	arRauschen: ARRAY [0..9999] OF REAL := [0.246739256236, -0.529170105611, 0.414309825378, -0.544103926825, 0.009949783811, -0.029587575492, -0.961653654724, -0.382605463343, 0.222026883158, 0.389023823093, 0.621050671571, -0.646958412688, 0.638418207627, 0.534061065662, -0.110754415353, 0.629669607832, -0.372363722573, -0.871060345803, 0.681706748020, 0.205129983440, 0.858041542734, -0.075593969433, -0.319802679147, 0.977319730903, -0.463662632934, 0.393306864076, -0.217856355895, -0.964407875275, 0.809210531413, 0.985531542521, -0.674619330252, 0.436784775739, -0.160868201578, 0.341967854837, -0.399787326721, 0.290907556563, 0.539355132357, -0.823844250498, -0.040486992077, 0.198136927055, -0.108719761440, -0.795757664573, -0.924329592637, 0.258815633556, -0.272619658361, 0.669346919862, 0.120580060721, -0.412226444472, -0.863110760094, 0.848406544850, -0.407508257473, -0.683558789495, -0.591427504389, 0.316833250828, -0.966288801701, -0.227470576788, 0.579664019389, -0.594067152985, -0.737773981554, 0.224918962597, -0.702529720677, 0.652896341734, -0.876627290498, 0.775098206896, -0.335284108258, 0.727377951755, -0.229819698701, 0.541187889029, -0.041203903558, -0.635223979412, -0.016835900977, -0.081127400735, 0.473800100213, 0.370010232427, -0.781292715531, 0.151475020756, -0.928262298559, 0.719073235463, 0.944742409840, 0.859713266715, -0.234696976409, 0.466709694464, 0.972663248100, -0.093433859902, -0.240648257108, 0.600574830997, -0.676848255859, -0.664059236041, -0.772492529238, -0.525769140900, -0.445967976269, -0.422592640425, -0.817647930030, 0.622493353226, 0.969345965405, 0.749765014787, -0.941528041560, 0.567473529861, 0.330423592919, 0.628163921603, 0.865778023332, -0.925525550689, 0.250234639214, 0.178032614233, 0.845317953168, -0.724431653562, 0.326294937160, -0.998925438332, -0.144238934713, 0.936006148019, 0.028752943103, -0.007566843574, -0.657885652494, -0.544697262441, 0.431807667642, -0.115466610367, 0.644197371225, -0.473158752747, -0.104897086620, -0.557304583420, -0.693084284084, -0.266431314125, -0.657718817527, 0.012733837449, -0.356939242672, -0.582847192411, -0.321250664899, -0.000437913139, -0.801730193481, -0.395392715595, 0.753309159993, -0.839167873710, -0.497709637142, 0.376142374662, -0.891710910001, -0.931460999004, -0.765244974856, -0.430077335395, -0.165793475662, -0.067370896287, 0.716185225145, 0.093961060499, -0.600848329188, 0.673058447165, 0.674704320685, -0.027227232800, 0.171745340627, -0.918910173725, 0.209163411102, 0.680797609799, 0.067226768430, -0.999009889300, -0.780625702217, 0.367241297318, 0.402204046803, 0.285102145157, 0.183271048762, 0.995194348284, -0.806487621398, 0.112997935460, -0.561176200081, 0.453177893515, -0.405486497721, -0.698964164112, -0.893396062005, 0.294927669631, -0.287540801977, -0.398405888092, 0.401119508788, -0.505326064545, -0.225827285260, -0.294225352090, 0.144798347025, -0.430384210188, 0.666149813029, 0.883918289765, 0.949635828195, 0.724396900619, 0.156010733086, 0.447585744588, 0.443566930836, 0.105623713564, 0.480873497360, 0.478874307928, -0.363553379976, -0.292587342811, 0.391116870080, 0.509282603531, 0.026478500049, 0.278623039847, 0.213444321271, -0.651644355304, -0.081057820072, -0.006698364322, 0.842760715437, 0.416093279887, -0.696197758558, -0.713828347366, -0.065887452693, 0.297891975424, 0.475395401787, -0.835706801589, -0.234477046070, -0.728620258748, 0.142537813675, -0.496592649012, 0.427164188114, -0.872643068742, 0.392931044892, -0.391015917539, -0.908629066401, -0.373314983099, -0.518141560956, -0.274306877176, 0.477171922966, -0.418180886710, -0.466110720658, 0.577632902938, 0.334027359560, -0.761070711022, -0.958568115698, 0.668176974590, 0.000497204020, 0.525722665811, -0.767668130265, -0.244392457220, 0.462184067229, -0.047276594620, 0.084864277025, -0.115062364457, -0.715907950963, 0.158290277543, 0.430925333764, -0.237143624360, -0.921853342785, -0.180352070779, 0.872419264731, -0.298218856373, 0.012398576959, -0.102073877969, -0.016164126855, 0.344215775954, 0.062456227753, -0.045480709999, -0.612235813695, 0.927440580288, 0.128274592282, 0.367175640002, 0.522036080855, -0.514356302852, 0.032995121162, 0.024509715061, 0.845448084989, 0.447884205959, 0.847428365298, -0.208174858415, -0.544927435342, -0.404805621403, -0.613620769868, -0.706941066657, 0.332305269893, -0.072931291890, -0.249740966904, -0.759240606791, -0.865256880141, 0.630348896703, -0.746062522885, -0.358926494928, 0.129871216481, 0.524777575363, 0.554834351075, 0.291634864464, 0.862406170075, -0.439019664257, -0.167620988081, 0.474524278117, -0.253399651970, -0.447962964225, 0.184329851673, 0.448599046466, -0.979074329430, 0.347509289836, 0.440450729671, -0.181101795764, 0.051759350663, -0.386345551805, 0.844407334874, -0.617550553980, 0.818452991754, 0.605805879582, -0.644762312935, -0.607126658097, -0.697909226410, -0.867331983037, -0.538829948377, 0.920977238585, 0.907194206181, 0.637867983590, 0.729978494237, 0.326346021492, -0.993639828643, -0.047669394639, -0.978448647461, -0.187853782006, -0.344460373153, -0.693377000027, 0.751878997091, 0.811489751365, 0.323523735780, 0.022615842344, -0.151697873914, 0.316030939885, -0.210096145889, -0.948333340436, -0.911576847596, 0.826438670365, -0.744203261189, 0.772633117720, 0.181996339876, 0.935860210219, -0.099340173278, -0.800545523085, 0.756346944715, 0.319694561318, 0.972386432025, 0.204278217384, 0.913860972173, 0.937730762197, 0.312294177414, -0.261802998374, -0.635043991959, -0.235704358395, 0.466866088657, 0.351908922889, 0.591241011493, 0.727184996899, -0.564588415423, 0.667864381168, 0.300950655987, -0.155187192446, -0.397009717286, -0.525668199483, -0.456722345352, -0.823156392312, 0.788091934648, -0.753677385492, 0.682613050591, 0.804545831956, -0.334143783172, 0.111262921985, -0.852217512624, -0.041248860227, 0.778424005231, 0.044092776273, -0.065148797437, -0.757446664925, 0.155584195178, -0.820895820909, 0.011012148577, 0.374346119688, -0.579777277082, 0.385402006686, -0.988425659978, 0.239650409460, 0.907806660527, 0.751302397733, -0.068518188527, 0.480588932436, -0.569440051514, 0.619651395135, 0.024224185726, -0.785251187626, -0.983163309183, -0.415107378772, 0.613246911220, -0.250774675569, 0.371154100200, -0.219976331516, -0.220820891629, 0.127276136859, 0.824871934223, -0.534679223208, -0.938731233427, 0.752572249594, -0.847763317363, -0.728473978394, -0.646685665337, -0.998230717786, -0.860355633059, 0.198309069301, 0.332641337457, -0.788086027259, 0.696356744821, -0.804116334097, -0.799940505629, 0.547771798051, -0.852007662520, 0.337985525103, -0.733625872664, 0.660112536732, -0.321721536287, 0.003955703369, 0.351169972261, -0.311372520781, 0.313518004463, -0.891545308924, 0.496612274384, -0.176333071866, 0.537443706881, -0.488325145144, 0.538839566528, 0.539455258831, 0.735078466938, -0.688582146983, 0.949128810865, 0.963534159979, -0.259586191929, -0.129749758499, 0.493600721045, -0.859039053261, 0.525898193207, -0.384840282320, 0.742109951586, 0.302311170266, -0.808430002728, 0.420777325583, 0.959985318514, -0.505694203965, 0.031473307543, -0.167052683511, 0.500995058621, -0.156240823058, -0.744660490876, -0.854345614702, 0.189686977569, 0.821968916196, 0.811848983783, -0.342248024788, 0.023386872211, -0.660481237660, -0.460544835850, 0.556515458246, -0.557324905873, -0.593178975950, -0.736410294210, 0.416696052525, -0.481910925306, -0.156710336625, -0.663890549795, 0.911054419764, -0.980908485241, -0.071421964265, 0.721864961899, 0.006623412636, 0.188458995265, 0.843334923818, -0.774386976596, -0.807321577917, 0.815744326141, -0.951120224240, -0.144390611699, -0.026540746706, -0.874864609556, 0.014619343280, -0.208958616452, 0.758626928611, -0.438345080326, 0.501296544538, -0.183694685477, 0.391828497818, -0.407011942600, -0.977859890170, -0.762130246845, -0.297107556927, -0.122704330333, -0.082888661982, -0.523983815486, -0.168575036587, -0.676178838144, 0.244686771623, -0.525082355123, -0.118407067617, 0.856705759830, 0.899986679545, 0.232731619176, -0.373659041440, -0.758853640143, -0.946684132010, 0.042597300244, -0.633489527377, 0.397335233294, 0.860053377735, -0.969386507574, -0.608982349462, 0.919627898896, 0.104498194003, -0.231531036526, 0.461295456936, -0.697220054250, 0.523414803843, -0.978859356941, -0.311641882775, -0.515670048627, 0.674862728618, -0.115816520827, 0.876629539024, -0.371659034411, 0.693339507317, 0.271248632601, 0.697480469246, 0.905967150449, 0.979868201460, 0.253258815661, -0.523955707108, 0.234763559449, -0.093833082248, -0.305544070723, -0.478107158023, -0.697737228676, 0.160904001479, -0.699222850226, -0.350695766840, -0.093324239932, 0.590288847606, -0.472075268771, -0.997304662950, -0.413944129832, 0.963282831881, -0.538669864124, -0.561804500270, 0.093857934354, -0.896970395490, 0.858943676421, 0.433641515365, -0.839191009984, 0.110506309259, -0.913682948113, -0.461490457417, 0.050243383716, -0.988280605990, 0.389764037791, 0.363904430651, 0.214157788563, 0.467709226526, 0.519997364236, 0.135818530443, 0.684759164261, -0.603702119034, -0.268419316193, 0.877117109797, 0.931384739652, -0.140717573327, 0.981671923886, -0.135246954639, -0.232401387562, 0.785244099903, -0.512140135299, 0.915155265966, 0.478784070983, -0.275938774048, -0.404748087264, 0.454006166650, 0.770802615119, 0.321755074255, -0.044838103921, -0.044766397818, 0.298751702852, -0.179385623660, 0.809437923947, -0.833841848312, 0.753779650674, -0.913838518064, -0.376044191736, -0.068730117317, -0.542593871867, -0.389049565052, -0.309568273925, 0.817561615928, -0.228143443931, 0.642328905857, -0.733360603876, 0.275236333669, 0.702112237526, 0.624421394323, 0.481857177133, 0.583799350677, -0.065337413748, 0.931548235238, -0.625969083958, -0.834512522213, -0.005650015820, -0.246010382853, 0.081298781207, 0.376488263004, 0.958702174688, -0.945974458932, -0.915934484488, -0.874287612394, 0.916799883156, -0.469450442152, 0.440713677224, 0.195323675413, 0.617040350545, -0.837318734479, 0.169952319734, 0.153771659724, 0.486478528275, -0.638819160697, 0.645997593065, -0.915354925421, -0.152165518207, 0.060295551424, 0.179416883964, -0.772015302469, 0.086118181691, -0.562826107422, -0.275447780295, 0.063906505211, -0.633526394653, -0.455850104037, -0.120851955932, 0.421106032794, 0.499620343209, -0.598850065060, -0.646616427358, 0.357237736603, -0.193854809814, 0.567724730445, 0.195663475127, -0.372821260522, -0.158056750685, -0.855837956202, 0.423096592926, 0.047027995341, -0.758922025278, 0.356971778983, 0.443647347943, -0.042147361226, 0.215564251448, 0.068340041183, 0.177291269390, -0.870104557139, 0.939236777196, 0.365008785213, 0.604158730590, -0.929579718916, -0.163665978021, -0.511346949857, 0.242462760136, -0.362591367359, 0.557188420226, -0.606221422767, 0.741195281289, 0.077036426793, 0.048193010512, 0.314666123135, -0.984858428444, 0.460746639204, 0.946057661354, -0.946166863918, 0.272900975827, -0.616788394308, 0.251179257590, 0.202353079566, -0.061445284179, -0.385572779586, -0.295799961294, -0.938227060849, -0.508337996617, 0.799743401620, -0.410014090727, 0.237535782472, 0.751036304509, -0.706447842465, -0.263237507081, -0.394747690100, -0.688150714247, -0.172462825669, -0.218692099507, -0.037766029401, -0.178199659551, -0.470927558837, 0.883228663781, 0.049918702856, 0.444438157474, 0.159857443072, 0.282221533557, 0.715223629573, 0.532428592597, -0.986489840111, -0.650364361217, 0.058543996800, -0.501009480370, -0.400235784214, -0.589280300995, 0.566421866038, 0.443685317696, -0.674411494955, 0.038062417014, 0.944215890637, 0.718572105839, -0.873071804215, -0.836357861660, 0.861249876716, 0.852403633336, 0.009361961914, 0.335102239078, 0.690320925472, -0.342135457788, 0.726486980000, -0.217484450717, -0.126917711359, -0.242431173859, 0.167341452212, 0.340963770653, -0.570551213657, -0.393229093423, -0.747032607878, -0.849476553392, 0.867814185849, 0.394966585026, -0.476517758907, 0.824517768713, -0.123745685474, -0.763511110781, 0.511435368053, -0.671460109581, -0.060036379791, -0.102884307714, 0.656986657907, -0.653404039677, 0.042770136203, 0.491850594452, 0.228272575543, 0.562898627376, 0.819041191154, 0.353312344924, 0.458881968727, -0.485155298790, 0.055094383845, -0.918719910364, -0.772592375745, 0.153732123944, -0.555993184464, 0.433087663116, 0.963410159996, 0.161010932370, -0.877731667709, 0.072961348815, 0.957803045363, -0.169325549683, -0.210430078261, 0.270182370919, 0.364976811671, 0.000887526570, 0.658057122004, 0.194342134023, 0.608790824187, -0.591578116787, -0.584628982855, -0.048320241703, 0.689196065412, -0.501091940331, -0.509502674411, 0.828689067846, -0.186360125620, 0.358118283074, -0.777402918788, -0.909671164058, 0.543782291077, 0.417043659840, -0.225356227100, -0.805139717432, 0.303729795010, 0.407044796304, -0.039811239061, 0.446407632663, 0.775584820949, -0.004740014571, 0.951315069235, 0.504543903117, -0.071948646061, -0.625458297470, -0.729660874600, 0.293493538124, 0.665903079080, -0.991178420286, 0.941126844696, -0.108546075344, 0.301003734455, -0.515422065553, -0.796223436435, 0.708593336614, -0.044071273723, -0.238737149707, -0.277276977417, -0.299167199866, -0.611572820793, 0.643683836363, -0.311036762095, 0.034698347125, -0.736555289597, -0.059452166273, -0.841744489550, -0.399957487547, 0.048641034050, 0.691121843116, -0.426142937448, 0.802617662814, -0.741494329790, -0.477954661499, 0.328158133299, -0.512215165726, -0.541295174311, -0.230194439432, -0.547034374221, -0.062024009281, 0.349314375953, -0.916724218411, -0.092744380301, -0.242786357167, -0.286735046168, -0.559148602503, 0.449041763777, -0.745158707512, -0.513680934139, 0.786026025783, -0.504750350939, 0.055350545515, 0.799483633198, 0.934405810138, 0.033922169696, 0.720637994545, 0.418491709645, 0.880158844967, -0.163137441728, 0.867818746018, -0.035334145941, -0.316515700042, -0.789617761172, -0.536104042001, -0.055134269823, -0.995597114343, -0.177001442665, 0.040769114729, 0.281875099989, 0.335676794887, -0.808991487370, -0.203335136870, 0.264173263606, 0.677808014455, -0.778769587235, -0.243410881675, -0.221057920766, -0.373071848858, -0.964506167651, 0.925577006119, -0.145365769285, -0.745957096826, -0.837329737556, -0.649573720357, -0.243767331016, -0.717820957602, -0.488103996047, 0.589287912555, -0.035391824711, 0.332107535576, 0.073973801950, 0.655044637327, -0.709540589187, -0.716071780494, -0.837772118059, -0.027656728571, -0.844827968721, -0.151940535527, -0.413167239818, 0.005011514053, -0.099245898407, 0.075226772186, 0.288592494403, -0.408640040908, 0.817498184105, -0.027674266586, -0.864782709192, 0.895092419611, 0.142483538548, 0.530743178155, -0.877081916830, 0.153623861285, 0.963376011897, -0.376765708130, 0.343760697511, -0.656038487855, 0.961393976984, 0.969850800604, 0.704099978064, -0.321644469795, -0.194963241375, -0.845246484367, 0.883097150948, 0.523139557285, -0.025904872022, -0.474928370917, 0.464591963031, -0.608894540802, 0.703450877615, -0.840748471231, 0.074940737279, -0.912829004070, 0.316523577937, 0.667685368412, -0.157405198168, 0.777038399599, 0.426964555419, 0.305664733153, -0.783179585430, -0.773095971142, -0.349441959185, 0.649764345670, -0.819401256290, 0.550662506970, 0.958334092391, -0.807662340887, 0.340864538215, 0.795147589984, -0.432285658620, -0.938935951697, 0.692164323306, -0.449196593529, -0.287304596732, 0.418878370143, 0.152337702287, -0.207140809159, 0.394871842309, 0.830431123909, 0.818073779406, -0.978273905752, -0.862804063048, -0.730298413145, 0.440110200389, -0.393436326766, -0.652877842189, 0.909220362579, 0.739095986019, -0.825817330538, -0.798492736161, 0.562865296033, 0.243296330804, -0.486844317404, -0.331653232697, -0.522004993936, -0.206970157282, -0.088377834029, 0.421952097925, -0.600802259125, 0.213859636921, 0.835919698579, 0.273560326920, -0.688558654402, 0.275055148223, 0.439068501528, 0.595496790447, 0.191442384332, -0.586591331319, 0.461177787306, 0.035502975523, -0.979483729818, 0.754914986795, 0.383257281124, -0.584778905712, 0.460985106816, -0.397540695073, -0.731321472446, 0.714271395786, 0.462776349401, 0.841844366225, -0.989997240947, -0.794638764199, -0.449690047504, -0.485538344668, -0.569066888656, -0.829496691942, -0.942956277379, 0.127429811264, 0.514096335955, -0.814996499054, -0.255271011683, 0.153170001235, 0.040702163574, -0.109755873757, 0.461556415658, -0.285080354765, -0.359789189277, 0.797148795582, 0.876352921004, 0.152166138928, -0.982440683952, 0.726129376904, -0.278422033739, 0.119560149915, 0.135627033629, -0.933593953702, 0.033842275089, -0.287177944145, 0.056212740374, 0.110418004794, 0.434676986715, 0.458408936391, 0.265619871609, 0.061257444881, -0.564588981038, 0.567841708280, -0.084344918771, -0.721688038706, 0.920242181131, 0.059390323772, -0.971319512657, -0.399220847061, -0.309027772333, -0.665363591489, -0.912709004152, -0.073862012407, 0.067684596554, -0.703681672957, -0.547543658975, -0.942830327682, 0.480511364294, 0.172985804095, 0.476793641540, 0.617990852035, -0.796430457935, 0.857861552747, 0.413594858525, 0.635925504248, -0.866751432050, -0.796863625788, -0.495670984759, -0.374977509357, 0.323023038392, -0.356534495453, -0.839284955030, 0.980838093521, -0.342406482293, -0.280793061649, 0.198936404862, 0.659048010334, 0.137553776046, 0.874818625813, -0.020766385024, 0.378235309364, 0.968067350445, 0.986534895183, -0.321368024193, -0.328216010417, 0.798171189457, 0.251190618051, -0.326446960048, 0.630696989342, 0.182914999951, -0.025160469998, 0.272208029527, 0.565919402934, 0.487738200483, -0.548172166662, -0.507209552389, -0.509070930640, -0.167269403356, -0.644923529584, 0.924804317692, -0.478564518226, -0.921762677181, -0.646762762636, -0.533560573390, -0.347591373899, 0.699635085442, -0.614636631781, 0.859517880907, -0.955001789556, 0.339146930192, 0.365286937025, 0.524010757265, -0.675270692697, 0.614162430227, 0.457875594387, -0.863092236849, -0.198092769343, -0.813516517860, 0.223903042725, -0.436347746362, 0.780841218584, 0.909398367207, -0.495892735780, 0.477911444061, -0.569395987579, -0.146650972714, -0.606544270858, 0.277434218151, -0.754911017839, 0.305274603827, 0.622224695243, -0.393998401653, -0.140010936742, -0.203988000067, -0.511531881327, -0.680583914457, 0.388166832955, 0.344343280756, -0.240779016581, 0.509725385335, -0.844520036211, -0.117103505839, 0.725892821341, 0.291263168269, 0.586311497539, -0.776273780858, 0.906667352621, 0.846415599943, 0.097490046589, 0.684382903922, -0.545299430629, 0.256859392073, -0.589408888082, -0.749586991425, -0.164804485149, -0.930954064471, -0.299620409894, 0.064335067790, -0.266619576663, 0.542000945586, -0.785794228124, 0.138801075284, 0.294517784166, 0.710127814010, 0.511363187864, -0.388462772725, 0.928953060587, -0.266970366432, 0.361628526609, -0.412034265924, -0.666934288741, 0.569230303885, 0.152134734222, 0.489457237793, 0.876157261275, 0.501140460733, 0.427246142821, 0.917589853444, 0.413867107697, -0.580480047566, 0.287150649219, 0.745621043427, 0.136538598132, 0.613800058631, -0.581144366207, -0.281306268550, 0.992292298765, -0.696688373285, 0.917588394205, -0.820359686104, -0.676661003820, -0.842408881117, -0.994234365810, -0.319103516201, -0.736723382956, -0.604760329980, 0.818239969710, 0.783820507001, 0.246185944115, -0.657196016149, -0.403697888127, -0.995150780822, 0.692288572933, 0.168061088419, 0.119921846627, 0.364989540303, -0.855680798907, -0.263656867290, -0.894865928753, 0.510699768994, 0.189185897617, -0.447285115440, -0.672978657070, 0.834544176670, 0.560712991509, -0.157172179788, 0.241893748675, -0.059960462351, 0.984749426453, 0.574429944373, -0.984005166876, -0.242616120460, -0.672194868062, -0.343482956009, 0.754578450154, -0.733255200807, -0.234196001373, 0.745137179546, 0.754168024554, 0.064314078103, -0.077932538635, -0.529696834070, 0.143181168371, 0.838996365305, -0.912757111243, 0.614893187871, -0.751880319198, 0.565478478436, -0.834012040735, 0.834466377047, 0.605493386525, 0.840176685857, 0.698476369341, -0.633077310679, 0.210397998923, -0.759788118676, 0.140552079897, 0.631965731021, -0.528836352059, -0.158802010956, 0.990369770890, -0.019803869168, -0.134520091606, 0.565686289784, -0.455613945489, 0.801903618746, -0.158640228982, 0.717202496622, -0.547831813729, 0.244780469968, -0.424876448018, 0.170836119607, 0.007398442955, 0.911729640675, 0.352723162010, -0.688599645402, -0.987557967310, 0.004866581123, 0.414027928388, -0.060997306452, 0.902315804242, 0.184449868194, -0.457073124164, -0.482700961612, 0.989282136499, 0.355302371863, 0.121561929992, 0.149376757201, 0.270869652267, -0.283803320000, 0.512882192147, -0.553083224721, -0.156770437985, -0.895244716044, -0.213404435345, 0.404663270200, -0.517802746353, -0.299143736385, 0.947496135212, 0.044415796670, 0.243940042318, -0.541746896363, 0.203075323992, -0.647373783849, 0.475455763212, 0.950029222674, -0.411124154545, 0.206910963904, -0.376899069888, -0.134490023804, -0.102678379475, -0.652690435762, -0.644841599001, 0.686166702982, 0.571332510414, -0.721995108026, -0.043151777450, -0.402344607467, 0.723838002602, -0.509802094526, 0.242244647607, 0.124710494179, -0.323613063161, -0.619797177647, 0.794161575859, 0.005887026618, 0.124043250601, 0.289828170929, 0.838632442156, 0.848401675807, 0.988685107482, 0.662462185339, 0.555603436176, 0.482507072074, -0.728481929026, 0.771618140088, 0.616755659382, 0.126330312130, -0.165651875853, 0.613194851370, 0.598795166672, 0.323378347178, 0.691073675685, 0.241795368319, 0.836520608106, 0.634843396184, -0.152796408955, 0.882721742951, -0.249667384979, 0.448022550928, -0.973888495732, -0.048223282158, -0.672215653461, -0.117773503850, -0.512046356795, 0.280992748897, -0.352288977687, 0.863336278769, -0.576514473578, -0.748917657195, -0.210550114103, 0.980285749582, -0.168263830413, -0.785262807662, 0.251342635236, -0.081944023883, -0.332136454106, -0.674013483319, -0.143140454083, 0.465366073487, 0.707227633844, -0.711361524552, 0.975868166976, -0.022668929233, -0.991241002732, -0.872139541534, -0.789547288093, 0.936903427925, -0.558566709390, -0.881144132504, -0.065177313557, 0.621683778496, -0.968916820154, 0.885734772176, -0.041834416053, -0.787493873826, 0.573085883964, 0.238603639520, -0.738198174414, -0.826107985500, 0.153163330451, 0.665122786801, -0.878637135620, 0.980801923490, -0.002578464858, 0.735024422951, -0.538046011407, 0.992437501271, 0.544194722860, 0.120774090982, 0.328717987111, -0.325934237715, 0.310302363315, 0.497984955842, 0.844682926752, 0.995588080079, 0.706294793319, 0.631210468099, 0.228669807408, -0.912198259278, 0.741572187780, 0.840490645130, 0.807003403287, -0.569320792578, -0.222549396432, -0.302197380894, 0.295157703050, 0.783764014430, 0.925797830200, 0.028125759206, 0.563416219327, 0.524987584431, 0.533081677544, -0.240901276147, -0.076048835313, 0.064541400487, 0.763086482722, -0.339499995830, 0.553329781541, -0.524726871946, -0.484614360692, -0.790739410342, 0.898061066711, -0.836621112100, -0.052849173120, 0.655469991192, -0.214857272307, 0.416654831582, -0.879289090105, -0.196311427502, 0.219039118636, -0.516144662974, -0.151080482903, -0.375475076803, -0.806263921556, -0.234486592381, -0.705077768435, -0.952567486624, -0.321264037957, 0.904525752713, 0.267993102165, 0.725670044857, 0.498733157019, -0.764168153153, -0.704535521667, 0.367409262529, 0.224926272022, 0.755633726790, -0.611155240728, -0.011822469637, -0.226443420070, -0.260992370867, 0.199083574662, -0.145859179995, 0.799470245229, 0.362667178751, 0.033129533202, -0.339480761857, 0.347214673992, -0.415584896701, -0.523249911410, -0.633641218267, 0.658197405226, -0.928007067246, -0.931473660996, 0.329023013517, 0.307743229280, 0.704663660831, -0.626125149822, 0.064110804330, -0.396204832950, 0.801903871555, -0.097628617145, -0.631229505017, 0.109477544147, 0.138394281780, 0.005201247953, 0.841772059774, -0.833261915977, 0.616793584946, -0.307703453644, 0.082269215373, 0.826023474865, -0.436379755104, 0.527494850768, -0.883648605540, -0.352355989442, 0.616470837358, 0.495010235917, -0.073042512843, -0.332992083423, 0.174980813821, 0.733407591094, -0.972981425712, 0.410256571355, 0.169312369902, 0.156418247668, 0.275844544789, 0.123441528773, -0.226397698474, -0.842374318258, -0.501579030967, 0.378505516862, 0.262934237735, 0.754730391559, -0.842646554643, 0.129130550773, -0.213984290482, 0.940937140665, 0.898425076812, 0.877111460176, 0.129683048927, 0.112619573848, -0.016998674049, -0.203358804152, -0.105409516709, 0.380551997523, 0.699146154357, -0.853907561880, -0.556377135749, -0.060995547720, 0.156334150016, 0.796882590833, 0.030625638650, 0.862570689092, -0.399004928216, -0.900505952037, 0.242665320267, 0.072634416701, -0.577841148906, 0.991618534974, 0.412447652219, 0.894287158725, 0.516298870238, -0.027424458257, 0.497612615365, -0.867438410611, 0.088002264399, 0.480835055999, -0.997299434752, 0.612839066465, -0.045010978354, -0.857028654135, 0.023685315190, -0.565765663427, -0.935541803692, -0.312356002636, 0.395692755010, 0.235544837365, -0.478605136567, 0.549637749470, 0.287108222598, 0.578706423299, 0.617358232023, -0.533641179307, -0.836487682111, -0.044419726777, -0.605437453149, 0.308625851764, -0.408431539811, 0.837881681701, -0.131970301496, -0.330951278823, -0.027217995685, 0.062031066559, 0.276185805806, 0.752827273115, 0.567123827715, -0.880712375155, -0.458528503599, 0.666317469887, 0.367683243522, -0.992320061615, -0.692190347936, -0.588289814712, -0.127162235633, -0.413428923381, -0.240580314805, 0.270494044155, 0.897600675575, -0.896485289470, -0.545190295486, -0.458514392469, 0.481797900527, 0.687154961858, -0.333094218352, 0.384330779443, 0.000997163224, -0.746776029283, -0.204979368344, -0.506025289354, 0.435517713790, -0.728484562382, 0.900071915062, -0.277351691324, -0.925994985457, 0.708026518596, 0.315979946932, -0.914501802280, -0.440516133774, 0.684116610812, 0.438736588470, -0.555057321648, 0.817167029587, -0.721478866136, 0.550485123819, 0.749501741039, 0.760924721584, -0.822565537465, 0.071643488142, 0.451132678320, -0.011098451720, 0.966005630119, 0.710873916763, 0.331784888220, 0.329672928689, 0.645012470320, -0.329369231336, -0.521326429995, 0.882773857049, 0.415501380069, 0.443521652747, -0.319963958358, 0.500104164757, 0.571514198096, 0.669833397443, 0.137664430061, 0.998124536845, 0.288839089218, 0.971864939383, -0.537123032358, 0.317282722826, 0.638681741265, 0.412217851427, 0.601306718188, 0.930870765906, 0.952487355328, 0.190335096749, -0.896484008243, 0.331142087312, 0.268061164931, 0.810019468126, 0.868362722403, -0.531867761858, 0.924499128838, -0.484451919703, -0.618806005144, 0.027564947900, -0.822881166742, -0.912712033556, -0.245611948564, -0.476086189148, -0.523714803806, 0.187417595035, 0.208248700883, -0.391706652929, 0.363413338869, 0.220018127130, 0.455549960662, 0.221071844738, -0.445751128023, 0.471516590826, -0.670060037350, -0.833973522562, -0.614770708193, -0.014785719374, -0.236502155334, -0.805653106047, -0.536265847215, -0.418059948899, -0.558454225871, 0.316677244740, 0.901364230208, 0.479343893527, -0.854761083767, 0.800365509509, 0.217316574883, -0.097844811381, 0.539709980393, -0.344316676413, -0.096972165160, 0.785891249467, -0.399645113207, 0.778003067365, -0.963470400404, -0.490585781078, -0.152794878701, 0.551272455272, 0.370518795212, 0.411997303300, 0.551903538887, -0.287627120424, 0.730690091778, 0.401823158807, 0.291065966849, -0.868441700103, -0.394679524224, 0.407878948228, -0.482070046802, -0.296957746500, -0.629025764275, -0.757295120576, -0.357254346020, -0.473807887941, 0.155022068449, -0.734000306702, 0.239137894598, -0.138023453394, -0.755265077755, -0.983738221821, 0.427266522866, -0.142703098504, 0.875734802540, 0.561284523336, 0.533652407889, 0.726277249059, -0.515189138125, 0.354648805890, -0.624167441447, -0.520751241180, 0.012887124529, 0.861682194802, -0.448597493802, -0.725291119050, -0.972181156280, -0.330987366240, -0.087314124329, 0.529654817424, -0.937182392487, -0.299131867253, -0.014385313716, -0.803442987803, 0.650981271709, 0.267317273583, -0.774024362554, 0.976640644489, 0.950527509208, 0.194620469760, -0.446446323684, 0.509252679484, -0.773597068237, -0.985717862060, 0.400509247767, -0.055843061452, 0.721705870716, -0.280102906504, -0.283297966306, 0.582302525870, 0.104755867780, 0.282993009340, 0.366307772783, -0.635685712668, 0.391824832045, -0.973496874962, 0.423374437338, -0.939957553921, 0.290751211056, 0.761116160615, 0.065792714802, 0.793381362417, 0.682918390653, -0.872450105669, 0.053809465224, -0.657846629442, -0.091401245849, -0.943840627973, -0.776392294691, 0.783480400436, 0.457753184982, -0.538907404730, 0.921450266798, -0.557454057608, -0.456486936368, -0.203885892925, 0.783758703346, 0.869736380141, -0.823051715681, -0.213523583162, 0.070586283643, 0.372630758246, 0.605570412378, 0.829600124785, 0.358163978160, -0.689409833684, -0.894752480800, -0.970190892186, -0.865856531763, 0.294132927303, 0.266001381890, -0.428342473718, 0.625749628079, 0.625214659828, 0.168773041757, -0.045151637353, -0.143866659964, -0.040999976241, -0.753874142049, -0.953132968795, 0.901823308848, 0.478045421615, 0.315547770523, -0.387898020010, 0.627537323966, -0.114666079525, 0.693745740145, -0.967798799802, 0.389862616052, 0.954346304157, 0.692881210580, 0.596993146516, -0.516819502657, 0.387843956697, -0.601677961988, -0.821941004038, 0.793138584991, -0.512097317691, -0.985022981878, -0.994159956085, -0.595393142770, -0.363379941561, -0.952011307263, 0.020683328926, -0.563677311888, 0.636349638801, -0.156300979415, 0.631929397445, -0.337343768350, 0.943833808880, -0.813420366238, -0.132074619271, 0.564184291531, -0.355161217065, -0.107640058514, 0.457258359495, -0.685956167467, -0.662267890009, 0.022791245298, 0.946210492834, -0.782725116282, -0.058541170014, 0.742354782441, 0.711387002074, 0.001971940610, -0.735200740692, -0.980084605884, 0.591697489030, 0.545792073385, -0.608610834420, 0.589834880296, -0.638251328806, -0.080026048164, -0.575913166490, 0.935533732286, -0.665266698097, -0.498579598436, -0.489433835874, -0.242752928820, 0.994636759478, 0.441254467374, 0.293993978343, -0.623006420458, -0.978083212395, 0.052289303961, 0.855611678263, 0.049539245226, -0.558413685408, 0.410609550021, 0.389848685235, 0.456648072255, 0.463209745653, 0.740506137000, 0.661382842914, 0.049067448062, -0.825265796933, 0.436436993445, -0.867666835093, 0.442572827851, -0.011924586643, -0.853639569594, 0.192740179786, 0.469032598401, -0.960778798569, 0.554163459835, -0.507419777404, 0.899184692481, 0.422368411510, 0.746641395157, -0.768038836472, -0.247406954183, -0.297322757061, 0.764798005450, -0.746197021799, -0.537788132406, 0.475280731633, 0.112577395711, 0.316289508268, -0.147624572352, 0.955874928072, 0.934960743230, 0.569409974796, -0.569903544072, -0.229482460897, -0.199279188506, 0.267784250389, -0.172149658738, 0.288559357243, -0.576918913418, -0.106415011254, -0.215563877712, 0.594860777219, -0.896107252095, 0.746421994485, -0.172439791402, -0.505989395998, 0.678987714449, -0.698606724940, -0.638020080968, 0.397953542661, 0.115732507795, -0.526264082654, -0.008893697041, 0.405671777952, -0.853374049517, 0.566690441169, 0.681015731894, -0.907219631771, -0.752308362007, 0.561964565841, -0.438930642705, -0.523209777532, -0.425623366096, -0.252875610982, -0.425537853123, -0.036259555074, 0.360943370385, -0.775496142177, 0.536602655882, -0.918951446339, -0.025465002337, 0.437781310843, 0.617108814810, -0.911880321788, -0.614325427366, -0.908644478958, -0.477000956367, -0.887235430672, -0.547570796481, -0.582256248288, 0.800134618451, -0.823655260560, -0.697010225344, 0.847147564270, -0.745080090541, -0.736766298561, 0.712284931551, -0.638476452671, -0.663306412991, -0.513065379943, 0.085093745579, 0.261154869869, -0.069953014151, -0.163370871734, -0.115964359095, 0.490289505526, 0.870832739711, -0.228134262167, 0.842811952933, -0.944686312576, 0.156353345290, 0.419239802880, -0.266552665480, -0.217474715523, -0.487866788299, -0.993337030761, -0.983394950267, -0.561736117977, -0.158810379635, -0.246798643079, 0.264992526850, -0.692275049838, -0.208427394755, 0.375107270753, 0.340045721686, 0.208101084644, 0.402941000199, 0.449856461835, -0.523059148547, 0.845476477519, 0.282890477033, -0.300200818448, 0.113847318539, -0.174350998881, 0.791928146638, -0.441681631689, -0.718734808125, -0.609926716441, 0.492771043682, 0.469401884038, 0.771186162238, -0.539872773385, 0.463663172415, 0.748568648538, 0.058006522201, -0.895954241288, 0.584796603431, 0.189667334788, 0.099025828375, 0.885762555732, -0.752092537832, -0.051509817836, 0.410052022014, 0.276549646818, -0.584315808608, 0.158826785765, -0.500260020888, -0.769170022158, 0.140054079334, 0.665432264888, -0.985382446235, 0.430303765269, 0.644821021677, -0.304121034643, -0.178494822133, -0.731644656481, -0.436776193388, -0.458229249647, 0.801286738261, -0.052083233307, 0.414391676969, -0.292116610246, -0.029555321762, -0.653606128151, 0.813512159153, -0.275858652924, 0.758697291033, 0.580590209082, -0.647485693191, 0.091811865407, -0.802885032700, -0.255262776367, 0.994806037816, -0.417402350604, 0.320392156078, -0.622899835974, -0.199253156200, 0.353650364927, -0.446345034048, 0.585033117249, -0.088809914775, 0.141828048260, 0.598579686269, 0.856373630416, -0.883530867659, -0.575325180787, -0.273900898280, -0.969173967753, -0.147944768110, 0.680762684118, 0.565467643004, -0.253416914711, 0.656011508658, 0.335778305737, 0.262623826536, -0.363422858420, -0.123545728074, 0.010148736665, -0.009640994079, 0.085687782316, -0.848163865207, -0.912217181392, 0.585102218633, 0.971079487157, -0.625911008936, -0.845504109095, -0.375672065870, 0.393710754600, -0.943235675452, 0.764443694028, -0.883314932434, 0.019400140511, 0.271814344838, 0.977770652855, 0.183268304081, 0.722054720121, -0.789626844877, -0.631077495721, -0.464411859889, 0.221670451947, -0.847674705566, 0.159232442769, 0.508595876237, -0.151644322084, 0.345180651002, -0.647616456529, 0.037864628454, 0.577454328119, 0.124833916808, 0.793593352099, -0.227381207283, -0.527758662493, 0.883026441620, 0.018435557218, 0.441465730688, -0.030964060367, 0.835687101698, 0.414300028896, -0.915581631351, 0.192463237369, -0.324749818510, 0.114849568880, -0.052509184399, -0.780697732128, 0.245685143764, 0.257953244161, -0.930958365845, 0.102876672121, 0.492713488582, -0.913710168168, -0.839988233365, -0.131755186301, 0.475983054832, 0.382387320431, 0.721128354761, -0.944108716318, -0.620414735364, -0.293768436304, -0.244052650611, -0.824448708073, 0.179730237111, 0.156744319506, 0.454341563629, 0.036968366834, 0.474860522376, -0.202214900775, 0.289185069015, 0.517731756737, 0.289272152953, 0.318853905847, -0.557790259095, -0.212559290267, 0.442897998078, -0.930741586288, -0.211732202860, 0.674534906493, -0.340096990185, -0.150897362347, 0.766187708095, 0.135545095095, 0.680977455438, 0.296029711527, -0.518360397274, -0.508875985407, -0.372041545714, -0.079329790693, -0.503482859534, -0.273641827719, 0.871522415867, 0.992722499594, -0.532478718920, -0.929288199048, -0.926841965834, -0.571456046773, 0.421384847746, -0.061966206852, -0.344863462587, 0.287453583722, 0.973042649507, 0.787018745957, 0.597701259818, -0.639521923642, 0.408962381559, -0.571436051375, -0.093153234186, 0.096920930155, -0.667142684182, -0.587548087729, 0.172375974790, 0.853852495882, -0.948302450887, -0.554620739254, -0.720522527625, 0.873786080581, -0.329519788682, -0.694419994940, -0.196550930888, -0.833208453327, 0.063800283076, -0.250087405464, 0.492599504704, 0.708285636285, 0.256604221710, -0.721652538005, 0.211437436825, -0.571728475101, -0.508100524096, -0.203081326185, 0.761565362164, 0.094253851107, -0.845800429215, 0.242160029523, -0.079797439450, 0.608635630713, -0.512627465590, 0.330476720965, 0.035027695775, -0.923136436664, -0.262454338411, 0.037095699657, -0.911438546901, -0.379149309361, 0.062161450911, 0.630316682982, -0.847029462417, 0.025722880242, -0.742454728787, -0.416368766732, -0.213037308386, 0.052029376076, -0.245326655541, -0.577418994646, 0.539414220259, 0.564101538646, 0.556918442834, -0.964365255716, -0.317608886877, 0.708956530686, 0.281445983821, 0.894253606223, -0.986857028576, 0.204991923033, -0.530022562136, 0.760818980698, 0.957197502345, 0.580063142741, -0.083263880916, 0.872385647125, -0.499030616238, 0.949064732946, 0.965250250853, -0.984533000219, 0.198431421811, -0.506541572375, 0.186837734550, -0.568574088924, 0.100636158124, 0.087016072196, 0.238286798084, 0.068084334577, 0.848449323215, -0.976802472189, -0.980236369250, 0.193509606001, -0.780313625526, -0.692272753218, -0.367577096129, 0.585856474175, -0.066823025103, -0.337695411912, 0.003583612828, -0.750419048676, -0.347317981416, -0.084210805759, -0.262602565611, -0.419728267477, -0.813362831486, -0.658877231072, 0.812790927160, 0.066417750665, -0.144599083508, -0.214575405332, -0.663173820551, 0.254724124749, 0.879760251461, 0.051138871065, -0.245129404155, -0.812324288700, 0.441234823890, -0.871664947518, -0.786364183243, -0.818901999143, 0.568845907625, -0.094976605407, 0.892471088731, 0.202648434457, 0.611718041268, 0.232413030401, 0.140828748342, 0.406546514860, -0.954527833940, -0.668369690918, -0.644070519622, -0.678245381543, 0.984248017186, 0.078896039180, 0.833272888352, -0.573557143853, 0.756607419365, 0.138381242066, 0.255969499943, -0.266258526106, 0.201234420627, 0.028140848996, 0.358254880449, -0.317557254812, 0.440303289021, 0.378584852387, -0.952905516058, -0.188179143671, 0.119195080410, -0.664080456653, 0.842134984833, -0.146587737616, 0.476581987654, 0.681867070589, 0.166220888676, -0.423342067761, 0.960136698100, 0.255280497044, -0.847295989036, -0.753668227803, -0.538058007570, 0.867213109676, -0.444339179700, 0.521418940877, 0.172740247956, 0.016771113449, -0.743035179186, 0.193129468097, 0.648796779284, -0.616611748512, 0.205730506478, -0.664329665256, -0.175132111820, 0.402564508979, 0.815089635276, -0.592924775308, 0.540059285122, 0.070423671048, -0.485932913708, 0.351875545151, 0.158036136882, 0.973949847883, -0.004067383387, -0.488272087426, -0.834686441455, -0.455405158240, 0.585903923958, -0.461918828031, -0.323396794681, -0.004123654419, -0.240004832394, -0.429659310129, -0.282033009737, -0.948452535244, -0.480648263448, 0.071155820194, 0.085662144955, 0.587287445503, -0.451812917182, 0.584527214172, 0.617659006305, 0.157683211976, 0.197815906848, -0.673834059840, -0.109004278124, -0.638489961601, -0.790740204868, 0.296319206590, 0.603497516964, -0.478040001515, 0.880845645216, 0.690785271037, -0.015887990584, 0.434041179478, -0.457946093064, -0.492608826446, 0.531282858890, 0.082890884740, 0.454745722198, -0.574266891946, 0.130927286826, -0.660983099159, -0.212288972951, 0.679272616204, 0.464687372800, -0.314278149251, -0.633935052317, -0.086231868932, 0.783019954172, -0.235243086481, -0.953555031517, 0.433993584294, 0.399391936248, 0.005964734562, 0.014957089514, 0.833298184238, 0.584572399937, 0.746830044177, 0.178822808770, -0.243488459463, 0.408530867001, 0.867152649598, 0.782991748581, 0.102010333383, -0.766718038925, 0.404637865406, 0.037293419044, 0.332821084971, -0.541231994359, -0.154206129049, 0.901772827803, -0.682734105054, -0.125796008910, -0.334096486883, 0.975153373418, 0.413872469846, -0.521738444860, -0.260782328915, 0.077398226970, -0.014761031608, -0.276124034060, 0.354936455796, 0.094732938102, 0.014749630427, 0.121989951888, 0.007338160400, 0.321607389407, -0.003308315241, 0.632721641711, 0.766663095532, -0.429080561653, -0.936243561595, -0.564125723497, 0.826124328057, -0.749600183764, 0.957080806195, 0.873841590450, 0.060859738742, -0.440430267271, -0.251931893570, 0.890889120948, 0.476525386055, -0.959517312727, -0.307549034695, -0.080979644716, -0.433967737449, 0.796393469435, -0.312701570042, 0.030346874059, 0.300877600101, -0.375539735860, -0.104899127393, 0.692697069407, -0.020706057268, 0.811179344979, -0.240720765864, 0.051442192320, 0.423146436546, 0.135542140174, 0.395203212158, -0.714241954082, 0.413072564566, -0.282279295215, -0.486403847837, 0.752315508351, 0.245472738670, 0.633102436322, -0.859644282553, 0.522452723039, 0.001357677823, 0.413217124370, 0.338333466297, -0.441352632961, -0.069252058353, -0.587057448220, -0.900981724873, -0.166152954070, 0.390893850412, -0.146100390955, 0.111504316646, -0.396131439352, -0.309777868394, 0.677289110823, -0.440046648055, 0.079836546814, 0.368222768588, 0.941803157443, 0.592602504040, 0.245852012369, -0.112086124723, -0.904421215161, 0.803391850028, -0.074107351872, 0.644117565599, 0.600003688139, 0.917980134188, 0.408432492791, 0.893543954836, -0.416565380996, 0.178848087645, 0.240638332920, 0.157808796480, 0.524950262223, 0.378476955400, 0.331852670226, -0.493056171350, -0.380468706151, 0.969272638449, -0.409588971499, -0.518481231664, -0.201723913988, -0.575833718517, -0.848257591457, 0.611467895695, 0.962173923998, -0.433975435787, -0.448542417344, 0.595948202791, -0.961493424451, 0.127906236768, -0.649011678976, -0.289470106241, -0.345819841171, 0.950061643064, 0.350311054571, 0.032219366377, 0.126401841113, 0.876105000569, -0.780471003514, 0.272305329971, 0.496728210837, -0.315439865164, -0.632732810241, 0.045970804162, 0.366851527665, 0.566165435869, 0.511518798875, 0.199534265792, 0.882749323673, -0.053875374663, 0.593870822260, 0.279678155810, -0.636850558528, -0.181981692157, -0.710002537442, 0.668312457388, -0.243649499080, -0.233611092983, -0.808181890154, 0.906877006132, -0.147317187877, 0.594202719946, 0.193383732898, 0.197855761442, 0.830811088498, -0.024450538963, 0.137947599050, 0.670805553118, -0.681669775679, -0.655662510245, 0.830803632697, 0.283147044651, 0.027630196018, -0.677985229211, 0.121460660359, 0.237685031139, 0.780812154907, 0.955236645660, 0.097029254828, -0.201309348901, 0.086328501209, 0.628515632070, 0.061065460908, 0.029277918206, -0.122669965291, 0.286225340788, -0.618652071004, -0.380995349033, 0.518830940503, -0.978304861892, -0.931976840624, -0.871115156692, 0.494478321197, -0.053673034348, -0.436579769424, 0.012527916773, 0.911076138492, -0.698066393477, -0.431182659548, -0.311197119348, 0.093555108419, -0.381882267188, 0.929709842248, -0.083438154884, -0.784122740243, -0.872912698630, -0.099484016799, 0.817560843536, 0.422018368019, 0.801616329912, 0.284808723346, -0.416975676864, -0.668425672967, 0.305260292711, -0.880778939913, 0.025061412116, 0.852556683710, -0.812715877312, -0.507117053479, -0.309907227350, 0.690020697454, -0.032974552207, -0.947756615674, -0.044965467034, -0.318958217787, -0.986008008558, -0.088679323527, 0.609238293668, -0.385532411783, -0.819133704364, -0.441838933342, 0.302507240927, 0.190043654248, 0.406884323432, -0.019841519260, 0.125064419191, 0.563511009961, -0.159615619862, -0.576937473182, -0.508679431044, 0.787469919809, -0.188103043481, 0.263252103771, 0.009747046196, -0.035110988687, 0.778099219772, -0.587237029042, -0.100000687206, -0.013678330124, 0.046504948162, -0.290742755651, 0.260039045356, 0.989893360496, 0.720505401382, 0.801915073016, -0.505020093129, -0.845173169849, -0.540693891643, 0.428409927551, 0.130243112099, 0.131828855959, 0.577628481553, 0.223962346080, 0.392711041039, 0.715074460962, 0.439333852490, 0.953962268122, -0.937626631571, -0.416639854631, 0.915871944344, -0.726148893592, 0.743016738846, 0.812062141177, 0.167579502950, 0.362096718338, -0.268949479076, -0.537555998149, -0.980685621693, 0.169475436515, 0.595501034961, 0.115678446426, 0.274319651887, 0.304705672249, 0.665791970325, 0.071193999338, -0.279339371012, -0.466255370672, 0.622337785236, 0.731570912211, -0.492042880480, 0.715588153984, -0.187833925363, 0.638539083568, -0.878605407776, 0.654885573091, 0.262926251809, -0.152047089563, 0.942012998663, 0.889501334493, -0.171622414051, 0.613740523470, -0.971450942268, 0.115554526537, -0.598533091807, 0.971336417264, 0.116086602424, 0.125137534612, 0.067045019857, 0.899482779730, 0.658483801336, -0.085137084606, 0.855714403262, -0.042614839153, -0.744186622785, 0.538868225347, 0.769292346827, -0.206284118877, -0.812724125207, -0.020116936917, -0.863426004569, -0.970363315099, -0.978038463272, -0.870562461813, -0.586041214128, -0.893394731701, -0.792746140913, 0.567832484668, 0.160323389564, 0.624321399175, 0.120808904846, 0.419353878909, -0.962567620827, -0.114718520660, -0.254397489930, 0.725890347845, 0.325826849785, -0.580176480750, -0.255053106842, -0.360012401224, -0.726060606300, 0.761507514503, 0.915504983344, -0.686553848078, 0.675884705801, 0.485927708703, 0.340640384256, -0.827941744326, -0.920298994026, 0.001134650023, -0.976973149916, -0.932132903124, -0.983818973018, 0.332159389597, -0.414240004962, 0.128168352908, 0.620630816316, 0.181516024145, 0.126376368177, 0.235006240988, -0.749671836845, -0.948954902415, -0.030369648709, 0.514186331569, -0.851015849233, 0.516973015512, 0.568439685030, -0.580950576622, 0.687792319712, 0.583458047012, -0.881060159774, 0.133571223846, -0.597943460741, -0.048491694476, 0.339563319156, -0.690737570482, -0.314172585132, 0.425146202831, -0.920816460911, 0.848775369977, -0.774080182916, -0.214723808362, 0.993465251408, -0.512643140985, 0.425261250196, -0.274627399951, -0.751921439609, 0.484082525362, 0.479018602430, -0.428597012860, -0.566255174600, 0.886287842521, 0.626553795054, 0.780318233707, -0.939240157563, 0.963669562999, -0.480937003790, 0.426534057831, 0.993047213682, 0.369971910517, -0.556436485416, 0.418529707462, -0.240708579362, 0.300918166634, -0.872560474349, 0.529723500439, -0.901596294947, 0.878874019182, -0.722168573227, -0.755325297204, -0.308410309688, 0.702739843343, -0.265119434536, 0.375711223442, -0.885776500953, 0.213093328979, -0.002388831158, -0.976908294007, -0.523097066641, 0.274242776482, -0.860746651154, -0.715232960873, 0.337270320046, 0.196693822150, 0.221294641868, -0.262675476263, 0.701200364841, -0.783545904654, -0.579192426156, 0.666788965692, 0.990334506218, 0.805348068665, -0.683525875334, -0.351526312508, 0.626950843270, -0.251621630132, 0.306250545951, 0.084506285919, -0.391355470224, -0.445595466018, 0.065286658328, -0.750623772116, -0.910007744180, -0.353621871153, 0.704328214192, 0.912638968658, 0.068871170680, -0.941273058532, -0.420794268164, 0.840961258567, 0.507448303598, -0.060571153458, -0.361498051469, -0.104555680190, -0.784237332282, 0.879242372671, 0.980673457979, -0.252936874963, 0.813677791952, 0.666987152561, -0.752891981272, 0.853436389339, 0.434817349712, 0.612948906113, -0.573119130040, 0.917707808637, -0.023133929820, 0.821373204869, -0.580251470738, -0.287730415564, 0.487565828275, -0.749667505740, -0.293098636462, 0.487402658230, -0.866648641397, 0.292096201050, -0.857000068953, -0.585865586437, 0.328612589389, 0.685553250262, 0.219530377071, -0.084724019922, 0.769364954510, -0.013173333500, -0.658075786906, -0.913704570926, 0.718088605007, 0.928295627050, 0.026117495854, -0.606840004305, -0.130012991090, -0.398775316214, -0.353776720611, 0.864207941430, 0.390126643877, -0.136040949472, 0.357457858259, 0.768212221008, -0.925987297236, -0.401987570029, 0.901733856906, -0.440716276214, -0.655771380293, 0.713999065696, 0.185445134957, -0.512142279534, 0.900481039637, 0.399866066626, -0.821247193079, 0.813524341226, -0.508714812937, 0.301306187387, -0.947882118886, 0.489043480508, -0.159809148034, -0.579992134538, 0.135903653832, -0.016724111656, -0.243989952202, 0.342064212434, -0.190849698424, -0.895578009908, 0.268341208123, 0.375792898103, 0.110332270584, -0.230688419762, 0.938089247766, 0.292522886864, 0.241154749474, 0.906104756774, 0.401506722777, 0.802746786045, -0.002758599158, 0.401547009729, -0.977396181062, -0.468334267868, -0.910754639937, -0.012037676387, 0.767950612443, 0.315341514609, -0.356932976688, 0.207563165794, -0.592027309835, 0.908527825260, 0.639726808819, 0.765898985102, 0.482240048470, -0.576581539154, -0.853408603146, 0.072949090518, -0.583525548835, -0.350193109046, 0.043760974914, 0.676704890144, 0.510193933768, 0.381768098628, -0.478911372010, -0.502168432028, 0.084562590324, -0.949159365719, -0.412302953750, -0.505502381725, -0.151956434949, 0.886272341975, 0.229534707724, -0.412036623746, 0.686439418334, -0.132301787309, -0.860129294352, -0.082177642959, -0.502397581471, 0.568352441643, 0.434947085084, -0.122553002463, 0.009850987339, -0.487674635905, 0.279841830745, 0.416706875588, 0.234422974283, -0.017420642776, -0.243523384153, 0.488149526100, 0.388982845502, -0.892408667621, -0.330965945608, -0.846572212355, -0.705954255785, 0.786604980582, 0.114206506073, 0.072772787831, -0.986347601873, 0.607593259390, -0.608140135029, 0.545616973281, 0.133792868009, 0.421492880020, 0.199327480645, 0.952200210293, -0.730455195195, -0.202768308399, 0.359731898190, -0.061177347196, 0.969933252944, 0.493063425134, 0.042543659904, 0.155143108690, -0.781490592372, -0.030592442240, -0.872042065395, 0.571338113443, -0.809227563677, -0.957975851780, -0.507499512281, 0.465735217018, 0.945942427840, -0.538597911441, 0.491857152241, -0.022928405478, 0.904743187853, 0.392389115917, 0.464124321813, -0.940430015610, 0.083335705488, 0.883009903032, -0.706133333445, 0.242451292415, -0.823493240016, 0.440544811682, 0.280812138421, 0.843494776908, -0.663452111977, 0.184603874897, 0.183810088781, 0.226642202544, 0.263911381666, -0.425748016003, -0.278113870563, 0.392146182375, 0.297931902449, -0.202289596397, -0.288004750253, 0.068626379918, 0.344531856093, 0.306346996969, 0.321932260856, 0.918002686994, -0.247605398966, -0.584293855827, -0.414442904289, 0.790490039099, -0.694150644077, -0.711696612756, 0.618266015672, -0.684577153135, -0.736940379014, 0.960651330266, 0.599937668863, -0.881828609626, 0.935520780064, -0.007709105956, -0.056382250653, 0.677864178228, -0.601887027621, -0.567272426447, 0.712658989576, 0.905867305156, 0.743734569480, 0.628472938731, 0.337437520920, -0.992036942765, -0.982283687165, 0.755407073540, -0.631490823868, -0.110057959660, -0.762329126389, 0.604316291599, 0.491238728499, 0.012360127518, -0.052599170083, 0.159818440207, 0.848481965993, 0.726475872346, 0.968552123522, -0.481428284189, -0.185599396916, 0.537129756527, 0.143325978076, 0.538166107223, 0.289772299912, 0.086098666695, 0.663303734678, -0.920524867458, -0.780218783026, 0.698024409603, 0.671901971549, 0.988244360679, -0.053415367075, 0.509581360489, 0.052405585490, -0.870610303723, -0.490542340198, -0.005741079988, 0.804774732365, -0.049909435386, 0.381428154224, 0.484369049531, -0.452141195259, 0.614620432654, -0.271435879419, -0.491422972072, -0.380607607530, -0.132895623682, -0.594715869989, 0.227843410632, -0.534035423481, 0.570610914637, -0.762585384786, 0.923057030623, -0.579043461462, 0.889043809311, 0.278100794380, -0.833828988018, -0.038546853490, 0.342664314655, 0.583074122635, 0.843975896603, -0.069149070206, -0.192017181631, 0.830254798490, 0.041489351180, 0.994100931796, -0.784511165342, 0.285235881665, 0.564327584150, 0.481225114949, 0.241871731227, 0.953320119991, 0.493024030607, -0.149801413883, 0.586726464993, 0.723551524383, -0.725431362396, 0.467464364229, -0.958214623717, 0.049505779865, -0.332405439762, 0.683175851669, 0.359616604578, 0.816472369831, 0.515375793652, -0.486530628766, -0.301768438204, 0.145118730849, -0.029368682747, 0.851499302266, 0.024803339251, -0.842986063888, 0.802541370561, -0.648125320038, -0.284782777870, -0.902795905558, -0.587388380112, -0.431681769164, 0.895725994813, 0.126505986102, 0.243096412469, -0.377777052423, -0.360402242320, -0.754791875250, -0.865504001007, 0.940937544760, -0.090586349377, -0.089144436389, 0.305644990483, -0.690637135813, 0.159694855191, -0.286813743280, -0.011401336919, 0.173486824129, 0.244155138806, 0.174998695039, -0.154802209845, 0.088335656643, 0.039399686210, 0.448355773203, -0.511767354976, -0.359220372501, 0.052811195029, 0.088739532774, 0.426121438821, -0.964157910434, 0.251909238412, 0.233241464770, 0.161138600931, -0.466251564610, 0.356817462827, 0.718234609572, -0.542914598145, -0.963624737337, -0.352104996654, -0.494878612916, 0.806253254956, 0.791764646333, -0.066203962289, -0.900299524979, -0.883339501180, 0.843074983483, -0.655824810727, 0.148313232276, 0.726615091858, -0.756856630824, -0.273480791627, 0.422202169239, -0.209549712236, -0.439235460866, -0.260234378385, -0.040857641008, 0.481177182615, -0.327401091398, -0.902456095289, -0.898735129280, 0.897159775688, 0.519332095319, 0.628440490333, -0.315692500480, -0.205765858585, -0.946661520431, -0.722176428984, -0.116532708074, -0.824289949827, -0.034870760677, 0.335860351559, -0.242791554085, 0.530143304165, -0.099711739022, 0.765875739276, -0.091692241248, -0.347646399816, -0.109887269630, -0.081365645688, -0.557353364449, 0.956928239733, 0.299169376129, 0.375221589939, 0.502233718897, -0.187203142991, 0.707388607526, -0.263978300249, -0.060533271377, -0.305328240654, 0.638532925073, -0.772015916094, -0.436099633563, 0.706256674642, 0.632384440644, -0.979219180904, 0.959492128287, 0.341082564333, -0.654837441661, -0.577112873730, 0.937929007379, 0.750762217903, 0.620066668192, 0.258996948129, 0.813175449012, -0.374435179002, -0.119854106697, 0.438754452850, 0.566006049955, 0.876647387571, 0.902366072864, -0.622536769207, -0.518452622590, -0.938399083298, 0.139331715119, -0.697296448014, -0.377674923080, -0.471512173245, -0.010737610554, -0.305889537142, -0.948768297064, 0.297842359777, -0.196435312685, 0.682507867704, -0.651304404411, 0.015536609501, 0.399253480107, 0.015716578286, -0.444073134796, 0.134847210838, 0.737569914516, -0.658402848731, 0.163789842389, 0.048429254860, 0.553855614288, -0.778510960024, -0.548605850041, 0.866781747297, -0.576970247941, 0.542838555445, 0.037664143588, -0.992439116925, -0.490017942028, -0.326384928816, 0.803426604811, 0.578748931220, 0.885780806870, 0.056989998234, -0.755267236574, -0.643688536415, -0.559757196032, -0.263016940582, -0.164427535437, 0.807378355149, 0.043332010743, 0.357995330178, 0.730803472633, 0.857347276815, -0.432199178821, 0.534348941454, 0.958167566388, -0.853020156120, 0.811333520058, -0.720452403601, -0.319378001163, 0.895290803133, 0.884787205622, -0.510233522980, 0.410427321999, -0.448989841951, 0.415116573079, -0.362664704029, -0.183288733578, 0.110178589347, -0.967460600020, 0.869970982219, 0.034181963658, -0.875277638348, 0.243050981721, 0.331259329166, 0.179851651380, 0.615638087541, 0.327857537570, -0.574292538438, 0.632085652478, 0.803815395975, 0.079001291726, 0.902509711713, -0.662130767397, 0.918107575366, -0.196268781737, -0.887647601533, 0.714303953224, -0.008834871352, 0.286744741674, -0.385489814193, 0.147076130038, -0.471620614307, 0.678907164273, -0.160728407772, 0.496218341883, -0.854219371486, -0.519599548842, -0.529584500236, -0.648174392256, -0.238623212362, 0.913833659088, 0.943307911981, 0.858399258579, 0.190599201492, 0.846713388021, 0.261276666765, 0.637218300693, -0.785872112831, 0.645388593233, 0.730735611989, 0.212443922226, -0.397330201744, -0.246861549905, 0.369428561595, 0.033306926978, 0.136070114941, -0.752173602753, 0.703998287407, 0.833339243631, 0.061964864910, -0.722752975778, 0.131848228800, 0.592270196573, 0.343581304450, 0.871265611432, -0.933150910407, -0.927984165602, -0.876730758582, -0.911842422455, 0.144605723414, 0.856243075656, -0.558412853244, 0.347791105196, 0.626833143229, -0.422055791649, 0.531989525815, 0.196161579780, -0.068730526830, -0.566396607442, -0.928121759401, -0.173120361847, -0.976744374836, -0.086405589116, 0.372102747993, 0.177462282114, 0.054967636779, -0.011020831514, -0.563562623142, 0.335943104525, -0.924956420232, -0.444745806387, 0.194495460125, -0.390884232548, 0.265089836385, 0.904832095001, -0.698233084785, -0.754368863855, -0.232397772987, -0.653692956321, -0.204155238771, -0.247446138212, -0.049111137982, 0.214184051898, 0.461168945535, 0.427679742954, 0.236990018856, 0.863524442720, -0.734838508578, 0.389244903548, 0.188774286637, 0.650832649709, 0.020754342769, 0.637825061852, -0.562449789059, -0.148833337516, -0.484530408924, 0.575624245590, -0.804399825026, 0.046795275505, -0.655384144157, -0.960585951428, -0.380319321736, 0.716843970972, -0.122355952906, 0.661126768039, 0.320949311820, -0.008929167604, 0.506344682752, -0.035140192417, 0.544398506930, -0.856712627609, -0.671723596803, 0.958787120943, -0.123047727073, -0.651137469119, 0.175355039839, 0.211603949629, 0.776787107729, -0.585520381827, 0.219603284516, -0.274972948126, -0.074642148208, 0.992571247150, -0.037231925687, -0.178986145418, -0.307128369001, -0.743153892132, -0.971984352313, 0.027848638189, -0.392267312075, -0.039080079436, 0.849867880473, -0.673337122527, 0.184827654345, 0.379615577924, 0.456597566895, 0.957638057997, -0.919376610017, -0.435677917232, -0.422108019803, -0.423234466762, -0.198913756754, -0.602184562228, 0.438519401845, -0.185147624194, 0.003714736967, 0.985451285043, 0.147134428913, 0.625980815274, -0.077729914623, 0.429083780227, -0.545014698712, -0.820987666107, 0.320382201481, 0.125830303235, -0.947958236051, 0.305362361756, 0.911706781239, -0.362515416462, -0.794242084264, -0.384642866168, 0.275975935727, 0.912683673657, 0.442810421029, -0.682807527333, -0.369255951670, 0.255218834876, 0.651414847650, 0.382217089232, -0.837850191368, 0.437870908168, 0.587572039208, 0.018297821800, -0.919107906893, -0.267792118725, -0.403484729859, -0.952012560067, 0.273488574239, -0.807810731935, -0.671616662257, -0.933407059252, 0.347108357577, -0.854169042876, -0.929284322968, -0.506233625742, -0.562840836282, -0.101734137887, -0.398117775908, 0.413944404853, 0.699148479895, 0.694581743036, -0.051667438309, 0.003666307723, 0.275814433872, 0.259110889771, -0.929268766721, 0.580244342123, -0.030379928988, 0.831708844851, -0.357287445394, 0.868513925614, 0.781094098965, 0.850141341433, -0.359300916892, 0.429415303187, 0.991338649811, 0.541098338465, 0.999407380283, 0.799379760551, -0.555292442108, -0.256737904557, 0.269537217148, -0.868634006098, -0.842874952464, -0.035924253273, 0.412061629776, -0.879821751841, 0.021487098927, 0.605081778479, 0.892268598800, -0.272647445030, 0.955660012982, -0.341744311005, 0.325545197722, 0.998597774727, -0.934990701332, -0.541196412078, -0.394452679817, -0.885844317704, 0.205737155866, -0.671023458824, 0.324211185179, -0.958802738575, -0.331117207258, -0.566716854326, 0.006826528234, 0.824265161439, -0.498209678111, -0.707127165855, 0.404062328753, 0.098456819956, 0.896006943055, 0.992762598366, 0.507016499373, -0.174668512794, 0.976009690985, 0.205978174963, -0.825906813923, 0.420043564563, -0.015084886973, 0.722260005016, 0.339123507051, 0.740363442692, 0.334873970306, -0.665231578296, -0.531058894431, -0.499557361182, 0.712053406926, 0.633096279236, -0.440664465585, -0.074669930083, 0.252039274937, -0.531647474855, 0.856838901795, 0.164644686464, -0.538880723098, 0.763826120605, -0.451597603487, 0.553912531247, -0.025642457301, -0.853175305940, 0.824665459621, 0.200711153287, -0.420366312115, -0.058603588771, -0.443903577760, -0.271072698232, -0.144299546592, 0.066272704036, 0.110271238262, -0.897656297839, 0.845572756426, -0.139497965328, 0.628413777657, 0.327996576962, -0.020983098620, 0.259219448598, -0.433907445090, 0.966916870681, -0.262781654296, 0.489220695097, -0.008939636589, -0.626873222413, 0.704588563794, -0.298833895290, -0.136949970368, -0.707363029640, 0.511221908217, -0.345818657187, -0.830940627043, 0.788046727273, -0.452653718538, 0.247720523883, 0.966669222443, -0.181314070085, -0.831476014442, 0.354085930487, 0.285518267935, 0.680040706892, -0.246571001694, 0.360554988758, -0.201042545824, -0.622707987429, 0.172768147467, 0.711740071491, -0.182729303240, -0.733004964153, -0.149417851669, 0.134039487036, -0.623197042973, -0.229152215222, -0.977810013611, -0.090722357266, -0.405297324272, -0.419064797822, -0.051445661160, -0.710063606619, 0.388654327932, 0.665033468445, -0.214022981831, 0.827872003071, 0.049047775868, 0.964078614075, 0.068166199853, -0.139999265352, 0.946906552537, 0.064789013609, 0.206864393314, -0.322275216546, 0.437951757846, -0.543388249681, 0.728598488933, -0.545265509287, -0.040472094212, 0.200909068123, -0.033136424039, 0.746004244670, 0.443593924862, -0.046006884591, 0.942324892925, -0.050580086212, -0.178037382679, -0.591487956873, 0.369507673983, -0.088141044500, -0.914147063864, 0.702535486004, -0.160105998080, 0.034950253857, 0.915751303763, 0.761858959616, -0.195043288041, -0.759970792809, -0.015864139137, -0.610283840848, 0.422829870771, 0.756298164321, 0.736992711524, 0.582888376358, -0.883049969590, 0.011300095195, -0.416519396959, -0.373919158356, -0.457671629297, 0.158779852204, 0.055769130420, 0.721676098778, 0.695031618402, 0.011677422028, 0.033987510244, -0.788571880246, -0.809749530233, 0.174417810779, -0.055627120280, -0.030203080212, 0.444696424918, -0.195197102433, -0.336103128164, -0.359043332136, -0.630966483598, 0.125554294884, -0.593242061142, -0.308287347841, -0.559988471094, -0.710270254813, -0.367561604352, 0.631529920726, 0.067325514140, -0.479089556004, -0.456053251774, 0.787020011825, 0.321938988708, 0.913670912321, 0.492211076523, 0.362574405294, 0.327634736645, -0.966252065632, 0.643944267006, -0.038677188511, 0.344760307127, 0.963178996722, 0.831541063284, 0.077157525786, 0.652742425532, 0.346352947521, 0.067890284646, 0.370654307547, 0.100680753759, 0.866043509237, 0.547320795998, -0.104086384403, 0.752160532306, 0.298598438906, 0.430541915847, 0.349718158748, 0.648213604577, 0.137830404356, -0.445449672236, 0.696419978898, 0.143957260984, 0.180303017333, -0.134923328237, 0.566492061052, 0.651600950366, 0.364256017010, -0.593378018260, -0.754853497264, 0.422554862335, -0.888479990055, 0.433289824478, 0.361871846519, -0.850051322784, 0.116258299378, -0.129872985027, -0.453980722024, 0.809890745959, 0.635669105250, -0.552723290217, -0.699644082632, -0.996578258180, 0.761725662572, 0.961237502051, -0.242687688656, -0.041306438332, 0.852514639401, 0.818195406514, 0.590456005567, 0.121041437154, 0.859468757428, 0.518590520983, -0.892427807119, -0.681856754430, 0.300962436988, -0.468050311787, 0.584432370787, -0.264299629501, 0.658356447289, -0.792049906313, 0.614927331899, 0.686544236434, 0.821781702166, -0.565520070885, -0.385076121439, 0.868794370133, -0.585446522802, 0.520525042745, -0.632951210322, 0.441053931515, 0.210453482115, -0.484019470621, -0.724755921474, -0.829635497371, 0.245232199104, 0.972895322151, -0.048023718930, -0.880315596765, 0.531946786317, 0.363534878958, 0.245649349231, -0.285801050316, -0.980176666660, 0.557307750041, -0.113743300339, -0.460376058971, 0.201093873437, -0.158521832351, -0.228190925153, -0.633136177253, 0.212543656550, 0.785587871650, -0.898449254043, 0.352334166111, -0.813716144549, 0.064756388280, -0.474296836611, -0.265382763124, -0.709837923509, 0.447454498794, 0.054523495604, -0.948191685746, -0.522482630491, -0.007329766159, -0.303378230774, -0.803330931894, -0.151676153877, 0.179893278534, -0.985358026488, -0.765369515221, 0.385330790913, -0.787161671465, -0.506170701031, -0.199811064859, 0.738746287786, -0.973081434108, -0.294023129660, -0.461794605730, -0.582557966319, -0.547466479062, 0.668447499966, 0.395597343575, -0.797233256828, -0.690878866288, -0.473996507555, 0.497249409629, -0.734394497525, 0.977686301885, -0.410536435993, 0.803000540422, 0.582257632406, 0.156630017031, -0.145001761042, 0.525278753000, -0.582788472077, -0.425680923860, -0.844919122500, -0.620874149351, 0.626122696541, 0.728573120498, -0.287187462139, 0.210411201315, 0.246953593475, 0.085605384866, 0.541343664756, -0.419656381462, -0.574230933978, -0.769725335778, -0.111526387246, 0.522929543715, 0.655816621120, 0.092451710527, -0.803900187952, 0.922369011277, 0.862073358728, -0.673054263307, -0.353494348031, -0.951598754456, -0.958144813196, 0.465578700108, 0.953749443856, -0.223513154314, 0.868120721336, 0.760180989446, 0.239463675031, 0.500735820160, 0.828752356155, 0.066488060921, -0.459891971245, 0.840879785413, -0.598337521360, -0.619060673169, 0.152275426629, -0.328102367913, 0.670274134615, 0.092770589522, -0.933258423973, -0.997412942541, -0.302799911736, -0.580090684224, 0.207631631737, -0.126723699097, -0.750620025074, -0.833561612873, -0.731161510703, 0.034274891599, 0.065571834544, 0.657352617465, -0.622566044249, 0.694147275703, -0.693393113445, -0.071705017802, 0.595762645632, -0.749046679656, -0.102769331874, -0.104937958810, -0.044852532485, -0.206591087515, -0.683589063523, 0.434129206270, 0.266940834884, -0.990019265762, -0.187074886493, 0.935293208500, -0.345469955546, -0.341320489763, -0.416614208878, 0.454876636234, -0.980796094028, 0.559360583708, -0.907823490732, -0.685949908205, 0.188814805420, -0.961385643943, 0.140855588460, 0.457392002078, -0.426631001016, 0.380769736733, 0.784791135071, 0.344519527230, -0.667203164843, -0.497152787871, -0.736085205542, -0.383288244011, -0.057288881366, -0.350089418997, 0.654639425108, -0.869441796883, -0.574876330345, -0.140934702431, 0.337105704283, 0.017857625488, -0.887669472822, 0.355796235989, 0.464187879485, -0.682515370738, -0.988101771589, -0.082147242514, -0.485982454465, 0.798674351589, 0.369543178987, -0.147047641434, 0.068506435511, -0.962061992197, 0.527301141795, -0.340664722440, -0.571293123440, 0.890705761348, -0.226895857139, 0.732833777022, 0.495013859952, 0.367399470053, 0.307938558400, -0.472720581789, 0.805980423912, -0.654302938177, -0.496508607686, 0.383492623932, 0.803124504730, 0.414640484176, -0.695628247600, -0.647357978179, 0.772107853035, -0.522825176198, -0.905371865149, 0.412478876628, 0.979243356783, 0.772666895470, 0.832364713811, 0.547222998158, -0.963136550754, 0.696183729478, -0.985647617521, -0.210334122503, -0.074111879741, 0.484489746242, 0.808998804503, 0.024900474368, -0.509642236008, 0.287784574492, 0.648544718592, -0.343064629290, -0.867945799396, 0.729131865092, 0.010667656409, 0.642902939744, 0.995039335500, 0.682970465921, 0.589024310956, -0.418846609953, -0.358916998697, 0.296143639074, 0.449288840665, 0.884103319225, 0.351746000311, 0.443768247639, 0.810443625548, -0.027510253825, -0.173347420375, -0.023682281152, -0.125237829270, 0.720374584583, 0.947049545814, 0.603759881967, -0.645694642590, -0.899942739204, 0.357637023595, -0.751981030460, -0.407638866742, 0.977696223337, -0.694455167747, -0.345051460328, 0.176407895036, -0.526732699789, 0.227705189689, -0.853087776477, 0.743085037674, 0.560762080503, 0.005821966236, 0.242050860553, 0.427647263918, -0.774659446354, 0.290537272807, 0.773228385029, 0.478858875800, 0.986866675493, 0.124644660952, 0.521777863188, -0.001874125193, 0.344226024693, 0.258665972919, 0.062818256725, 0.695133995066, -0.881537899992, -0.121676541266, 0.846078155695, -0.336738496528, 0.565296741815, 0.469949546164, 0.554620808839, -0.410567835346, -0.787315144663, -0.190685602141, -0.998921441171, -0.907700683516, -0.875633743483, -0.027373002259, -0.437468212877, -0.094709794450, 0.054417120547, 0.497927453788, 0.353342670195, 0.381461855105, 0.182397487159, -0.495416003757, 0.248608415396, -0.687753647467, -0.217660837215, -0.612400102465, -0.409880678940, 0.850982098026, 0.237712243488, -0.116224241795, 0.008380569063, 0.458457484611, 0.794826020712, -0.969375689306, 0.410275246674, 0.774812782737, -0.155545323140, -0.714503264939, -0.730519796546, -0.854069772865, 0.639571412793, 0.774470456828, 0.748143897207, -0.593101503131, -0.894596697011, 0.737690644469, 0.785884340981, -0.691769457167, 0.761525819377, 0.337794363021, 0.352747845070, -0.991375573648, -0.713420921979, -0.407248585488, -0.444000888265, -0.827053296421, -0.970250284623, 0.363173489430, 0.046720735138, -0.586845311729, 0.161139268736, 0.534598146501, -0.597195504528, 0.506971366743, 0.573798602183, -0.599356460422, 0.249921705928, -0.463193310308, 0.986343950626, -0.677032460105, -0.510225244604, 0.460346104271, -0.130126875894, 0.852343329174, 0.748021566129, -0.220384080422, -0.987874289997, -0.909281284486, 0.168058802106, -0.661627977487, 0.032234075620, -0.025846669567, 0.237774329420, 0.807562152095, -0.599412130559, -0.507643532380, 0.837591869465, -0.831764963669, 0.097930515051, -0.378171409127, 0.758198851913, -0.774003335410, -0.300685164730, -0.517723696387, 0.117881488648, 0.561770049451, -0.287290211782, -0.572933510598, 0.218277722924, 0.673122918492, 0.293886853624, -0.736618889689, -0.804262933501, -0.921253909782, 0.243305710420, 0.516514646785, 0.338523894557, -0.115666174033, 0.857505872463, 0.645077669452, 0.533696719142, -0.509520372635, 0.255062509836, -0.376862090442, -0.954011308597, 0.715250283542, 0.615668387775, 0.385145388157, 0.604189843502, 0.889186366710, 0.464144894529, -0.779375073869, -0.875171262655, -0.705428534035, -0.743880166957, -0.679909690455, 0.466411600730, 0.269732288079, -0.246172381774, -0.728640396354, -0.194564482571, -0.429113833480, -0.674083882703, 0.645568422673, -0.919714023380, 0.609937633441, 0.835577327977, -0.158326371712, -0.825629041169, 0.844293857641, 0.127865659026, 0.536480534164, -0.194081547513, 0.466372233055, 0.837400093620, -0.550133350084, 0.644928272013, 0.980054578394, -0.703165458952, 0.616826192150, -0.661636007887, -0.572011246402, -0.284441438663, -0.493006945230, -0.604681519330, -0.398277269900, 0.897930044790, -0.779667957571, -0.099468848671, -0.731693494071, -0.778600967306, -0.746947501775, 0.013298683075, 0.967240464116, -0.854138961220, -0.300176787889, 0.147708891042, 0.629164415799, -0.707181140891, -0.239637335855, 0.859783862161, 0.713696762701, 0.977450182295, 0.164361186815, 0.321300780653, 0.118359755353, 0.730429786721, 0.614516762543, 0.962875582364, 0.239129695188, -0.980452229297, -0.160277221087, 0.554842095662, 0.423386363237, 0.765125654793, -0.241233558073, -0.046018331964, -0.837404605948, 0.174183698568, 0.108247285849, 0.567868547428, 0.194380523743, 0.336488160631, -0.269249609285, 0.697373584593, -0.478245715876, -0.002143830762, 0.058687856963, -0.863630753462, -0.594603479519, -0.783945944454, -0.386510635957, -0.598893606896, -0.213080359833, -0.261970092352, 0.832485676785, 0.707413030605, -0.941494842278, 0.737214525840, 0.459142123020, 0.802912114605, 0.731894365983, 0.151830624315, 0.702973091773, 0.986842129797, 0.782696821660, -0.964774564907, 0.952710851456, -0.078345155492, -0.860889007480, -0.224288795866, 0.458028730934, 0.752119609682, -0.027976677031, -0.236139028068, 0.484973045006, -0.198797694713, 0.472615206082, -0.713512361051, -0.854046922948, 0.512585215117, -0.995322331005, 0.434964778257, -0.006324783038, 0.161976486949, -0.670644291856, 0.478073697739, 0.279769773662, 0.276655156300, -0.489783337131, 0.488891448552, 0.589696086975, 0.890374390164, -0.852174905113, 0.736268024772, -0.966241502292, 0.491020060260, 0.706788421794, -0.595331187027, 0.274827723102, 0.666513648724, -0.723606000948, -0.235739966225, -0.040027823899, 0.612552722139, -0.066844230714, -0.444459931479, 0.326502881594, -0.735352130049, 0.790577595330, -0.095273208764, 0.811678690925, 0.401560932083, 0.355093655620, -0.245645097166, 0.280608164256, 0.974715558210, -0.862017879065, 0.569738852809, -0.476878306978, 0.947509414229, 0.042828378748, 0.041624311187, -0.803977709379, 0.252608986315, 0.749524095907, 0.364650790337, -0.116237831384, -0.651140677602, 0.510237133066, -0.042187506659, -0.603066402230, 0.179518978294, -0.104505453853, 0.936268722393, -0.535601746798, -0.602768254185, -0.055185108478, 0.879204171213, 0.140626825206, -0.940629397527, 0.047627009889, -0.233555583431, -0.157206041208, -0.261610758369, -0.151019462428, -0.567541106599, -0.314017221178, 0.873578065756, 0.911581105361, -0.225850457363, -0.296097548404, -0.191727560123, 0.775314906648, -0.821543015065, -0.973125413447, 0.112803166487, -0.613167446329, -0.481238493425, 0.075485522266, -0.833410036806, 0.703049280186, 0.359466055084, 0.987384315399, 0.781621644288, 0.998208282930, 0.818696008243, -0.449444525998, -0.698536210946, -0.490853665425, -0.142076155931, -0.080222025573, -0.541670127968, 0.146624468585, -0.874896440720, -0.829575942534, -0.700844437277, 0.893639294486, -0.225967075178, 0.677187446045, 0.112736952375, 0.596167233877, 0.602453605272, 0.993171055172, -0.292313024453, -0.145519138616, -0.611883989785, -0.421100110906, 0.388295576500, 0.986022009872, 0.569840528144, -0.199196155250, -0.605632847555, 0.363070718499, 0.778842333622, -0.579971121915, 0.299711573199, 0.667941982636, -0.170022112411, -0.137138571307, 0.563715808256, 0.468277506121, 0.551308811789, -0.995251763206, 0.785526353842, -0.204656135665, -0.128336829198, -0.898399738134, 0.757430309565, 0.758442270058, -0.999595143355, -0.051592644421, 0.742566569897, -0.451961228155, 0.781591999702, 0.185982473785, 0.831392206427, 0.654954809704, -0.808983140981, -0.021254365645, 0.166031371878, 0.298759761691, 0.660465970926, -0.986196889081, 0.032189886905, 0.717173322756, 0.478414361998, -0.009806480942, -0.643121305963, -0.961350791939, -0.644751964078, 0.266935627368, 0.718148787351, 0.511597608008, -0.493987152833, 0.910584861477, -0.585170983525, -0.478099607316, -0.954472992117, -0.047205846212, 0.149319295576, -0.643791941421, -0.248251744628, 0.612433061857, 0.001260889739, 0.545750458305, -0.432732093988, 0.021350158645, 0.099161027751, 0.686662814309, 0.340070390405, -0.663657612035, 0.861941555120, -0.375605539733, -0.486416300341, 0.354272977602, 0.965379536110, 0.093416943650, -0.848880669927, 0.494404725089, 0.143270061513, 0.140519970352, -0.119214477540, -0.269323083652, -0.070946937807, 0.002907497033, -0.453234835676, -0.220653223199, 0.083186162401, 0.329206910743, 0.719905241317, 0.157908287257, -0.021282074727, -0.474242921472, 0.860764354344, 0.911756182634, 0.771762797366, 0.188363208997, 0.815790449871, 0.177570909368, 0.578336488243, 0.609279225856, 0.874328550760, 0.388224811136, -0.522250706711, -0.401744996688, 0.097473362812, -0.344685729843, 0.166086123633, -0.991141693145, -0.977369494276, 0.208857900733, 0.167117821447, 0.697547647984, 0.502446928517, 0.052817317412, -0.717627844909, 0.395781561303, -0.191736490958, -0.466008853534, 0.565190009421, -0.666692381995, -0.163997807315, -0.774034501495, -0.914461328557, -0.513024659233, -0.964227291634, 0.978890048768, 0.180182761242, 0.103570027900, -0.178412501503, -0.447777637558, 0.666880428996, -0.188093410103, 0.048934996491, -0.524491625232, 0.343346064503, -0.189004169974, 0.123734753485, 0.732152432322, 0.259177067312, -0.809538449828, -0.498203420988, 0.355247676148, 0.710083464514, 0.800950361799, 0.472569627261, -0.290935265222, 0.890295298712, 0.066524231003, 0.162471498398, 0.300231586238, 0.945776496147, -0.439026836139, -0.221246580332, 0.122774879191, -0.225531334474, 0.387624499361, -0.891291657771, 0.188582836190, 0.098676115900, 0.096369198338, 0.893502456627, -0.296045822849, -0.061742734575, 0.113443331251, 0.282112530097, -0.000297086084, -0.720862430500, 0.101996753148, -0.198035779735, -0.671930680254, -0.399648179021, -0.067578341974, 0.929542946885, 0.419300333807, 0.947822294915, 0.039944923043, 0.706115813909, -0.206876044814, -0.304014774491, 0.434560512111, -0.727703472113, 0.436106977132, -0.304142741507, 0.217669423204, -0.085556585072, -0.851975539416, 0.441069940113, -0.228303518991, -0.578812598941, 0.104886204412, 0.200428480288, -0.197084808642, 0.935440914632, 0.122257872725, -0.903656974078, -0.106268077594, 0.914529447330, -0.336483188548, -0.874751327571, -0.968267646673, 0.089864973805, 0.886889819347, -0.459846434855, -0.487928354200, 0.377409655742, -0.790062441958, -0.118332491706, 0.040839525865, 0.775769335757, 0.725601626704, 0.331015473618, 0.834469141004, 0.455731246665, 0.003359188767, 0.701678698806, -0.184440894232, 0.629364634253, 0.835914761660, -0.309544823334, 0.642502214395, 0.963661595930, -0.393090847087, -0.818060194567, -0.203923046561, -0.658171240539, 0.839601712101, -0.369768824102, -0.874937873018, 0.971733856042, -0.737820299025, 0.785289658356, -0.240550457600, 0.376820874223, 0.968422122396, 0.843961376927, -0.365730113794, -0.689804825832, -0.181075158991, 0.070172527311, 0.092043710164, -0.788151760915, 0.013190049560, -0.976604960396, 0.732121547976, 0.385531225280, 0.709150034137, -0.102455423869, -0.317430259939, 0.497228981202, 0.428311591989, -0.056225341073, -0.100915600448, -0.278695226313, 0.384846701183, -0.985003758378, 0.456092849293, -0.078917325981, 0.650750452068, 0.673417882580, -0.009215355933, -0.909047559910, 0.573419889610, -0.957647463389, 0.313146151525, -0.432639899655, 0.254205464817, -0.346786500099, 0.454342032100, 0.421429733829, -0.585025209485, 0.822706231549, 0.317861747235, 0.630968726938, -0.180278615320, -0.201569850578, -0.813207218705, -0.759814214691, -0.435224833611, 0.927858571533, 0.041421372319, -0.966285864225, 0.481352682244, -0.961999935238, 0.290286128953, -0.899569165198, -0.502574279610, 0.359427865183, -0.031624333159, 0.288287249215, 0.462710369393, -0.463027857103, -0.451886455258, 0.186873710240, 0.815768748477, 0.428883299100, 0.918505023240, 0.020008446470, -0.006895851890, 0.453504952488, -0.413963002115, -0.988507553578, -0.447228559187, 0.393909284357, 0.683275381008, -0.822873981232, 0.152198357181, 0.256268212902, -0.911009527893, 0.733337314570, 0.791603346694, -0.496718654549, -0.156193342378, 0.578852524258, 0.970200002313, -0.342499648225, -0.350401981192, 0.766784655629, 0.589326008440, 0.384454328718, -0.169778053740, -0.464768610497, -0.039176621566, 0.755543703403, 0.513907180583, 0.318790648432, -0.935806960171, -0.668674375071, 0.433934253747, 0.302058439564, -0.116784689002, -0.336809456579, 0.465739784627, -0.949219505529, 0.709651235894, -0.223089809436, 0.483325302347, -0.864002542128, -0.049551835466, 0.818198207136, 0.281571197818, -0.603737054694, -0.037828717286, 0.605125666244, -0.195821700067, 0.384459650056, -0.984172398255, -0.647086899211, 0.552666004228, -0.537490918767, 0.351201066363, 0.812508304075, -0.791900642013, -0.793767770295, -0.683753092849, 0.236399083956, 0.357718115871, -0.151910022765, -0.009636611892, -0.517849472468, -0.887417426681, 0.051500900782, -0.453237446664, -0.772304878026, 0.828538441986, 0.718157705538, -0.957897676777, 0.111205255689, 0.827605632447, 0.694104872741, -0.998426626251, 0.807593153363, 0.024550130559, -0.698901819154, -0.532126049618, -0.808802005078, 0.578582861808, -0.586291804425, -0.118008629716, -0.658546225128, 0.810887369323, -0.601138654162, -0.520380278451, -0.624167870612, 0.339104064379, 0.305036265023, -0.052271810241, 0.123834447041, -0.485704911498, 0.086182027517, -0.983094742471, -0.824596434192, 0.817117929061, 0.102553800997, -0.070549092115, 0.293827869718, 0.900492018659, 0.293277640226, -0.370325978524, 0.965639220652, -0.299000928041, -0.070262154531, 0.503414264947, 0.244727090985, -0.519698573287, 0.462481776802, 0.829843347635, -0.223752299271, -0.781240027099, 0.661148504378, -0.395794881768, -0.659048193325, 0.220123575649, -0.727623320757, -0.398498056404, -0.130500064312, -0.280868367065, 0.151796340391, -0.427227289686, -0.770292784066, -0.037339491188, 0.948082056899, -0.316764024755, -0.346498237131, -0.668737381433, 0.933778061800, -0.035292081338, 0.168418527691, 0.614856995104, 0.294896835062, 0.715472004862, 0.727892849526, 0.482979883278, 0.726311850377, -0.824015748997, 0.395727106675, 0.619324124110, -0.568031910438, -0.056952991298, -0.142780968472, 0.535111891738, -0.761096290442, 0.390494208836, -0.951889188443, 0.973344991711, -0.004289207926, -0.727153371395, -0.363442517135, -0.452341298726, -0.028845366427, -0.850656973902, -0.288745448919, 0.255534015838, -0.414994082980, 0.971456215853, 0.234764846290, 0.244580774659, 0.016946185676, -0.345453826360, 0.300646224193, -0.373695008452, -0.952467475057, 0.101530671042, -0.735274046472, 0.112948494565, -0.370981978481, 0.199552563554, 0.103966668042, -0.858110455956, -0.758590331513, 0.454798940095, 0.169947962905, 0.626760444085, -0.174077658915, -0.176089356115, 0.386054070417, -0.456802474006, 0.929038164579, -0.905295644546, -0.786870893900, -0.908338733676, 0.059032552493, -0.739842531841, -0.744599870159, -0.515548047486, 0.686999258210, -0.487415515552, 0.862825609194, -0.658601594749, -0.113519347145, -0.247750035711, -0.828186022916, -0.624660404694, -0.902381889198, 0.027499366566, -0.388697633894, -0.441438813751, 0.025585914334, 0.507492205257, -0.823478389606, -0.405413777253, -0.951801024372, 0.267615944721, 0.450732552456, 0.195186424997, -0.972693789609, -0.934399130040, 0.502816994205, -0.749141101710, 0.285954279548, -0.098609162217, 0.794214279491, 0.414916167158, -0.600179396943, 0.425925090851, 0.139184689502, 0.208314922602, 0.598111427859, -0.031380788663, -0.514193097575, -0.170716331501, -0.589154471155, -0.859923986979, 0.063546590320, -0.297807630291, 0.608841220173, -0.980950972648, 0.123007026733, 0.259020486268, -0.180568178881, -0.302399258939, 0.723066450623, -0.114619092596, 0.597744336325, -0.342111527727, 0.766565338186, 0.324064931320, -0.344165747063, 0.620309690978, -0.343969614569, -0.098917308409, -0.327893514340, 0.021653999396, 0.451646093330, 0.526129559729, 0.791139887411, 0.997245806810, -0.849531806269, -0.722456817376, 0.120149362994, 0.564075194928, -0.972804847013, 0.791463366507, 0.585382326704, 0.599213791927, 0.948472401408, 0.049328312221, -0.261593646522, -0.637322369527, -0.901751704074, 0.592804459306, 0.990941515888, -0.587670708384, -0.480042898168, -0.218361677066, -0.445561377483, -0.107641834781, 0.890984691453, -0.356055971983, 0.745835502747, -0.733417499547, -0.088781275761, -0.702753780637, -0.089130579021, 0.839008919209, 0.524634170126, -0.759472239430, 0.816601038381, 0.770508129122, 0.843350401344, 0.326937319483, -0.416325500283, -0.298625198739, -0.298396134984, 0.824110169740, -0.539388203126, -0.335787553471, 0.469685848075, 0.143926726588, 0.201649924844, -0.054738586520, 0.133030632149, 0.943346004186, -0.259811322380, 0.675334981776, 0.732210826170, 0.672074080853, 0.673776954560, 0.919468039292, 0.771171987092, 0.157652621441, 0.771416084839, 0.837566959318, -0.464260752808, 0.669226995260, 0.855837485121, -0.737509518270, -0.787825900517, -0.350632462712, -0.110487644789, 0.337866627418, -0.466137167436, 0.750562965590, -0.122819563699, -0.841878499551, 0.669883109535, 0.810150279222, -0.760966508423, -0.566116889960, -0.548415992847, -0.026513190270, 0.121240795569, 0.646346135720, 0.398873889852, 0.116867265423, -0.543176484564, -0.291153813962, 0.796694477743, 0.336196163681, -0.197051932652, -0.040828521116, -0.141307410588, -0.617840691108, 0.598842823356, -0.153765641233, -0.946957806948, 0.781062652147, -0.287803776551, 0.097611656219, -0.557611553722, -0.102294527573, 0.782124202565, 0.288934581116, 0.368919409083, -0.361168536066, -0.282481662672, 0.152416303635, 0.939603146931, 0.130514119329, -0.648161361842, -0.930315090765, -0.891810685377, 0.572878860332, -0.379683468253, 0.556785178770, 0.722622594734, 0.243895461269, 0.000352429748, -0.075922645978, 0.289395988362, -0.322199733950, -0.362692434170, -0.752931983456, -0.003051309962, -0.728157720773, 0.395864443725, 0.410454166903, -0.493232764290, -0.988751477142, -0.216531967015, -0.200653211420, 0.227335960776, 0.926548388844, -0.606757140647, 0.537806812271, 0.259463319804, 0.256488982598, 0.262858679721, -0.000247842740, -0.096928444960, -0.627873306491, 0.877911062594, 0.411841948079, 0.167364656590, 0.358851237259, 0.797028813254, -0.150377135875, -0.773586834960, -0.198348888041, 0.029381186560, -0.184852327600, 0.505147655158, 0.894128912678, -0.263167179957, -0.233246746854, -0.218730181315, -0.199530201814, -0.861614800290, 0.293693041716, 0.252735887586, -0.892054594487, 0.684286250691, -0.520875244497, -0.969573491349, 0.349993412947, -0.341340467043, -0.985219516267, -0.273612885400, 0.591655920623, -0.581238181840, -0.617191745324, 0.260869848744, 0.327940179466, -0.212187970969, 0.402973846259, -0.789528533835, 0.093517467718, 0.360362947111, -0.288572536422, 0.012025584826, -0.370270670495, 0.840597684634, 0.509976598769, 0.554548785523, -0.473962750559, 0.301929014893, 0.454631332102, -0.792118195964, 0.809946483280, -0.126163887511, 0.113792469231, -0.866190187540, 0.060486758794, 0.583033758573, 0.003625319835, -0.470207469430, 0.792487993990, -0.788475657671, 0.530913907804, 0.877022683936, 0.236690690349, -0.392075451569, -0.016275032083, 0.375219998578, -0.428936429619, 0.108263415867, -0.455352562830, 0.774429742103, 0.225643964518, 0.543846044697, -0.998401632232, -0.686416221054, -0.898503876146, -0.686050811092, 0.432629814097, 0.344885229710, 0.206173750389, 0.929957440166, 0.857227065110, 0.805112882594, 0.723001444125, -0.521302678163, 0.577008512431, -0.095372135527, -0.811202736494, 0.503928565450, 0.432234333520, 0.236037728017, 0.682256459268, -0.375487344313, 0.716607195367, -0.810389959258, 0.294026209302, -0.807637029534, 0.397024025607, 0.539356069750, -0.217447983756, -0.709497044943, 0.451041078344, 0.924418061293, -0.031107745411, -0.747034010697, 0.589198065339, -0.291903033965, 0.728253240307, 0.890620073890, 0.540816947977, 0.550644896217, -0.342017980135, -0.670663574889, -0.477750425756, -0.738945714187, 0.065217382758, 0.169394026158, 0.841637373437, -0.908768241584, 0.367294876897, -0.546062690868, 0.693389326770, -0.751286256093, -0.331404180956, 0.135153628365, -0.801092848887, 0.919002427642, 0.624010579849, 0.425502316009, 0.350449833585, 0.061009372302, 0.099800001601, 0.993287417991, 0.737209836832, -0.535837867636, 0.034125130899, 0.156394877137, 0.982973785856, -0.398241151949, -0.579010863098, 0.689268749364, -0.532496797526, 0.525898437661, -0.274198098042, -0.583195691559, -0.696183488099, -0.817371788824, 0.222981024408, -0.483172142120, 0.466282074405, 0.008882673524, -0.131079104155, 0.305912068794, 0.346562867230, -0.371031639173, -0.981149021988, -0.928444678280, 0.101456688604, -0.462813332818, -0.838500710324, 0.829054066108, 0.985720437970, 0.611242309073, -0.464357923618, -0.674153187561, -0.192530681552, 0.438544414233, 0.685373490761, 0.600405218730, -0.495553295147, -0.004522862694, 0.743974867321, -0.072170910710, -0.894792424086, -0.984911135249, 0.925435355699, 0.170730595304, -0.180742323803, -0.814156856075, -0.161111205879, 0.869644270672, -0.438152490179, -0.509781575321, -0.070157602628, 0.603642139609, -0.729017498606, -0.770035847219, -0.960355558161, -0.793199523768, -0.444814959562, -0.381132747657, -0.480465563476, -0.752855749037, 0.875707801322, 0.623886943634, 0.647242087476, -0.573252035392, -0.182956250830, 0.381331589099, -0.441667425279, -0.526508979236, -0.065186681266, -0.022148619790, -0.839414750958, -0.516672105165, 0.414452119419, 0.764426301633, 0.711466535968, -0.367034841012, 0.743090455445, 0.459451190775, 0.014242450039, -0.921423637909, 0.107421569013, -0.796758195655, 0.483448606285, -0.314602793100, 0.352485789289, 0.175936626738, 0.571912647241, -0.795264895587, 0.433462515493, 0.153825623293, -0.717933521857, 0.508444148994, -0.455613863785, -0.746113750441, 0.054908634461, -0.886243456651, 0.255790683215, 0.043271113084, -0.009706801493, 0.852113479974, 0.547775951077, -0.186682192658, 0.990284323782, 0.417291064733, 0.822840597929, -0.800554812169, 0.689310808095, -0.515196841432, 0.288729392905, 0.330993092959, -0.808893481831, 0.098993315260, -0.569336035631, 0.078313954835, 0.068368708233, 0.226028130585, -0.116020482862, -0.614866474938, 0.431212394733, -0.745051989764, -0.911009110322, 0.837306705086, 0.106191857553, -0.952504593436, 0.177071027851, -0.992317847491, -0.412091306254, -0.672074256095, 0.059824314839, -0.490948831881, -0.269702657605, -0.068639961082, 0.822517086977, 0.752564831912, 0.760622981079, -0.707425621467, 0.312405058502, 0.083190413266, 0.792638523621, -0.756200284938, -0.879244471476, -0.195239691940, 0.383343732991, -0.893358552759, -0.430885060450, 0.426719852409, 0.376070675620, -0.736098293059, -0.421597610790, 0.828002783678, -0.101009062745, 0.715570759224, -0.040091414275, -0.575083073210, 0.130843012597, -0.819088841468, -0.098287652194, -0.122855408288, -0.300602358841, 0.299666804370, -0.902027162924, -0.441162972520, -0.689692368573, -0.293111380662, 0.042521979113, -0.591178998913, 0.971795479105, 0.993041377832, 0.091063341756, 0.870576538732, 0.685991402537, 0.647093345850, 0.198009901778, 0.938877413160, 0.467457964971, 0.745773561831, 0.544318834423, 0.791264032651, 0.791564822474, 0.766901376248, 0.589401496897, -0.785402228383, 0.864233281056, 0.787101774956, 0.919643744694, 0.119406513335, 0.478566894363, -0.609474668648, 0.995440576006, -0.405669428661, 0.718955710643, 0.413253057896, -0.450253026964, -0.266205572221, -0.246578840306, 0.849621617099, 0.446917459212, -0.319244023056, 0.357719768604, -0.270767252166, 0.804409666683, 0.636106430940, 0.119476480567, 0.265185417675, 0.772344808215, -0.034506862558, -0.713336390118, -0.898489609675, 0.304309023651, -0.223964114094, -0.432187192604, -0.992814781810, 0.055749207419, 0.121101894500, -0.831064289089, 0.980510462962, -0.316083075394, -0.630119470863, -0.995575220382, 0.532058068961, -0.606447253801, 0.454736804858, 0.166577954401, -0.175266958072, -0.713279129315, 0.756827717210, 0.625070499234, -0.809966267951, 0.794026470789, -0.798686754922, 0.894026906522, 0.823148236690, 0.341112936614, -0.232567754473, 0.834145895501, 0.667313608290, 0.218233792255, -0.780655801191, -0.985281366803, -0.451558964603, -0.393921417626, -0.613329493816, -0.876466187592, 0.699249782578, -0.376402627902, -0.797573111256, -0.786226842290, 0.701693738499, -0.521124669259, -0.911324558136, 0.604054270972, 0.600912902342, 0.221052753248, -0.425989325266, -0.246047470854, -0.114217625354, -0.794262657335, 0.170697842508, 0.469878973019, -0.542248697924, -0.777063638550, 0.898985958348, -0.812308876593, 0.490561580135, 0.308255760675, 0.152299094039, 0.713520613183, -0.935507159759, -0.120055429364, -0.535651274649, 0.117235377383, -0.947823566780, -0.564765386391, 0.246383281253, -0.775684508211, 0.422922862863, -0.513660940638, 0.861968381319, 0.205125859841, -0.737269952331, -0.916594154019, 0.085339444777, -0.030615384822, 0.595294589721, -0.453624616486, -0.302094257251, -0.164359887143, 0.209732274787, 0.390428562987, -0.152146540887, 0.598149045068, -0.495852953267, -0.166344271782, 0.841945744430, -0.448200840342, -0.855567684658, 0.093344893905, -0.626742858787, -0.321965329564, 0.358005199181, -0.379110339677, 0.377919029304, 0.592206560042, 0.504462166009, -0.341249206990, -0.747052900237, -0.524387318910, 0.737104617521, -0.592132329113, 0.776223973392, 0.348789248336, -0.556858148402, -0.169145602897, 0.993977734720, 0.558087830669, -0.081801008590, 0.932860845102, -0.325257323904, -0.561312341190, 0.270879319124, -0.349021831866, -0.545422925951, -0.013073491449, 0.391810613615, 0.422601186184, 0.754017380607, -0.846185489212, -0.717519125430, -0.954827048913, 0.493336756838, -0.349552269400, 0.480710031618, -0.692244757648, 0.187643262191, -0.796173322439, -0.626705108629, -0.802968985760, 0.714684347996, 0.190839541937, 0.441637323947, 0.887246004534, -0.793181286339, 0.293196107334, 0.592358743249, 0.570150056013, -0.367871058398, 0.336461603877, -0.333277619662, 0.070981003510, 0.992426660558, -0.043647392206, -0.484123307755, 0.363525336111, -0.614253474271, -0.426205229675, 0.631881198273, -0.298638677620, -0.268036847705, -0.423054161413, 0.165154796387, 0.308424898771, -0.650656527784, -0.612768743542, 0.737688665230, -0.729535441941, 0.317360263080, 0.735201595085, -0.016717156118, -0.369603090677, -0.541953578866, 0.027986340162, -0.103629668477, -0.352646575941, -0.673914795122, -0.986356723872, 0.279563191842, -0.881205294201, 0.997572352478, -0.952778556570, -0.592202282915, 0.948439161204, 0.092989274133, 0.759936990981, 0.408172407373, 0.331407111535, -0.648703546765, -0.379065801481, 0.876978314400, -0.466668340681, 0.263555177930, -0.368224380866, -0.431862566027, 0.879134355801, 0.444002713083, 0.373569051461, -0.158907048296, 0.690507764498, -0.102769774868, 0.076972414128, 0.668978418792, 0.906685205639, -0.430808163389, 0.126988531224, 0.920745352689, -0.701733012976, 0.751100548138, -0.203016638666, -0.566355730381, 0.823969221183, 0.684969151064, -0.528900917521, 0.442005477868, 0.002069652395, -0.776331615381, 0.063132907062, -0.448090215790, -0.404401478031, -0.485450515473, 0.734746445405, -0.035207448196, 0.143078922423, 0.553486826607, 0.239998614283, -0.910974447150, -0.850344707164, 0.643725091047, -0.502680562577, -0.505612864371, 0.742846108170, 0.313202825279, -0.551526439816, -0.565330285473, -0.894290814421, -0.398904014753, 0.124711791627, -0.346924557440, 0.115176730272, -0.218095862376, -0.221888488575, 0.804116712809, 0.787210030682, -0.920250146781, -0.400742663483, -0.737685481963, -0.419636040504, -0.148673590047, -0.006671811739, 0.820199426532, -0.290330073625, -0.634064561444, -0.042981274109, 0.587893619311, -0.612867202143, -0.351580914328, 0.154846507818, 0.787926334934, -0.731147569270, -0.904492254604, 0.971260203138, 0.756653088821, -0.253187596177, -0.091001673861, 0.919657576420, 0.860637307736, 0.924060576060, -0.307669182982, -0.383545441630, 0.879346780343, 0.078223782307, -0.567494709146, 0.904980710530, -0.413730747462, -0.891908642631, -0.978038543673, 0.387893678594, -0.325473085993, -0.303269931997, -0.290551008627, -0.365144321250, 0.162515457865, 0.833640035392, -0.634104300498, 0.749469022356, -0.355830506758, 0.704465607246, 0.531262595892, -0.289047361855, 0.536131760541, 0.945997995501, 0.973375019296, 0.311988095210, -0.048883994870, -0.622975837781, -0.046716138700, 0.221677258747, -0.817600890959, -0.805434295382, 0.280347277352, -0.218890765458, -0.886967069571, 0.694706861704, 0.348140038671, -0.727407956341, 0.786417902504, 0.025627728876, 0.523679069552, 0.095350220366, -0.660370754283, 0.429118635108, 0.598847062057, -0.962432184067, 0.229611044675, -0.884381638916, 0.507025316799, -0.037321449901, -0.327728023583, -0.278033902026, 0.516268158483, 0.579938696459, -0.156481061487, -0.207417486560, 0.429990815736, -0.493792301060, 0.391565012139, 0.198199578816, 0.379526838310, -0.754868840211, 0.169597051629, 0.194534738656, 0.583020070755, 0.113117485815, 0.600900164791, 0.094472366517, 0.843199423088, -0.836297397829, 0.215035544286, 0.420870035157, 0.964958034972, -0.594208210613, 0.918673895429, -0.038241571124, -0.871206296241, 0.666680500928, 0.581742941258, 0.053387683824, -0.637367710766, -0.033547447810, -0.522166975680, -0.741485149469, 0.396252574280, 0.821192629945, 0.922382857977, -0.174603137023, 0.534818202144, 0.876463959677, -0.346767496559, -0.734258380497, -0.934669949641, -0.871560147106, 0.348540326780, 0.212731437432, 0.858189970840, 0.198476495641, 0.260968885704, 0.882535611708, 0.378603238158, -0.295228202021, -0.869066404405, -0.325627817502, -0.031289385958, -0.544709484809, -0.477816372068, 0.282892781637, -0.538185002761, -0.575933611498, -0.744023236771, 0.889936551981, 0.903826594738, 0.195012043924, 0.342567180047, -0.088603714662, 0.564985480663, 0.452910903575, 0.562841044065, 0.576898336935, -0.976802734837, -0.721367356122, -0.253975332740, -0.872026603023, 0.568019115545, -0.577853715178, -0.444147033776, 0.417787843855, -0.390486450087, -0.663814376992, 0.612636518710, -0.059175953836, -0.638269385808, -0.899459898322, 0.748269080014, 0.762814040868, -0.518249944278, -0.623094223539, 0.788217839965, -0.504720811330, 0.502142632969, -0.956412343441, 0.313174745258, -0.794448997183, -0.615621929956, -0.260797801349, -0.285756460966, -0.520630468843, -0.815150904551, -0.006069695953, -0.555854460011, -0.311898807327, -0.633654683944, 0.949531474260, 0.511676359192, 0.288384536229, 0.170015110948, 0.487956361032, -0.074268457630, 0.677840719717, -0.819187858316, 0.534628685187, 0.298501323829, 0.248960241327, -0.849976401943, 0.502678566169, -0.338210203854, -0.214835934670, -0.046192481363, -0.183406914297, 0.439560089200, 0.945175245747, -0.621388699335, -0.761036742491, -0.868347665877, 0.097766390132, -0.086335449868, 0.812920245026, 0.299438436242, 0.118376929556, -0.713349613721, 0.910281721984, -0.381388105565, 0.626724887499, 0.531330067315, -0.775774849332, 0.613740772365, -0.542230094097, 0.336278029460, 0.928740307566, 0.852877232610, 0.925654165913, -0.043509730919, 0.162145307660, 0.049688530877, -0.529966341249, 0.828762946066, -0.444099517771, -0.526810398839, -0.869364625822, -0.561645194517, -0.524427434520, 0.375598529956, 0.118978765436, 0.602888445966, 0.417138608829, -0.552384431758, -0.855901839193, -0.128062565022, -0.181885652742, -0.562286056215, -0.013038824776, -0.627073878702, 0.617416934012, -0.690335131315, -0.141403985118, -0.844165678447, -0.085046780367, -0.857487379902, -0.480349530414, 0.862960419408, -0.271628281051, -0.713344127288, 0.665220449080, -0.775096683512, 0.625108907412, -0.566586693860, -0.833320021995, 0.450677973731, -0.210327503577, 0.560922311073, -0.849298239162, -0.906109677232, -0.107808144637, -0.265958007436, -0.988442229158, 0.716496466241, 0.402011895588, -0.803563258824, 0.470143826106, 0.592962744830, 0.868104240232, -0.221860129592, -0.846338201702, -0.285851553691, 0.022983609419, -0.968521266215, -0.720661016391, -0.248798867568, -0.388253680108, -0.910224366450, 0.709107520301, 0.874846296583, -0.097218620477, 0.691467355004, -0.411062884682, -0.443589089591, -0.055912784874, 0.251481509024, -0.863352891632, -0.273466715800, 0.205230991902, 0.355250774850, -0.367273991377, 0.315052524646, -0.376811066407, 0.441536426806, 0.666673515070, 0.774747979523, -0.803824095169, -0.544614079983, -0.674752436865, -0.990186534847, -0.777075929332, -0.664212673696, 0.212118831218, -0.287918470411, 0.230642890654, 0.228821550934, -0.526586947784, 0.554887828184, 0.134090130435, 0.800504421721, -0.919975491030, 0.741903072896, 0.374742083384, -0.188027571002, -0.973096113988, -0.856722467554, -0.442382751272, -0.286584654460, -0.574940499045, -0.549361590850, -0.528559916434, 0.890413536148, 0.061105408017, -0.412529122729, -0.604780360952, -0.937803248305, 0.315131324501, -0.690964212587, -0.448678301162, 0.280735657066, 0.508889683902, -0.431900654088, 0.645260992170, 0.906911396535, 0.326900763787, -0.456232139135, 0.399229996980, 0.040199047652, -0.811624136219, 0.925858434127, -0.297748927113, -0.511182178088, -0.131324027153, 0.591431597609, 0.025426909664, -0.025464790644, -0.358913623685, -0.311722424356, 0.004996598122, -0.247682459959, -0.159153253552, -0.781405106458, -0.191513758559, 0.181389294640, -0.380046685288, 0.075100692017, -0.769567212398, 0.616459565349, 0.069719997224, 0.414443149537, -0.150128310370, 0.258334021168, -0.188764294719, 0.406784569104, 0.336207263744, 0.379152245055, -0.829222865320, 0.608685552284, -0.740390529902, 0.345861132218, -0.911407856540, 0.011643053441, -0.927787920196, 0.737461335912, 0.803292196392, 0.154555946373, -0.766504442782, -0.585810434411, 0.491909560028, -0.684196796305, -0.699244023956, -0.768887623620, -0.422726385657, 0.918364328576, -0.006570803163, 0.024451855455, -0.402296616214, -0.874855088110, 0.624798103832, 0.849813038636, -0.178848384816, 0.423014149766, 0.966616120571, -0.918251658703, 0.685134572647, -0.648350486213, 0.640886702061, -0.063819098551, -0.711066709988, -0.973148805007, 0.191184684512, 0.798168364498, -0.976670923339, 0.040225308905, -0.643658528537, 0.285770496810, 0.109127879355, -0.178343780682, 0.477133203801, 0.948341407018, 0.320470492395, 0.742755661449, -0.792556155036, -0.820504711094, 0.292041690729, -0.850681747980, 0.258977974144, 0.166755718650, 0.511894887702, -0.201120158834, -0.145210404237, -0.079075049459, -0.695035248158, 0.694744140541, -0.460964008021, 0.760848756424, -0.052084898365, 0.545235984041, 0.174319262931, -0.463152358387, -0.436334583991, 0.346830141731, -0.894063944239, -0.054062897766, 0.356917562822, -0.651655437199, 